(* IEC 61131-3 sources: StandardFunctions/iec61131-st, 18 files *)

(* ---- arithmetic_functions.st ---- *)
(* Definitions of arithmetic functions defined by the IEC61131-3 standard *)

{external}
VAR_GLOBAL
	PI_REAL : REAL;
	PI_LREAL : LREAL;
	FRAC_PI_2_REAL : REAL;
	FRAC_PI_2_LREAL : LREAL;
	FRAC_PI_4_REAL : REAL;
	FRAC_PI_4_LREAL : LREAL;
	E_REAL : REAL;
	E_LREAL : LREAL;
END_VAR

(* Calculates the square root of a given value *)
{external}
FUNCTION SQRT<T : ANY_REAL> : T
VAR_INPUT
	in : T;
END_VAR
END_FUNCTION

(** Logarithmic functions **)

(* Calculates the natural logarithm of the given value *)
{external}
FUNCTION LN<T : ANY_REAL> : T
VAR_INPUT
	in : T;
END_VAR
END_FUNCTION

(* Calculates the base 10 logarithm of the given value *)
{external}
FUNCTION LOG<T : ANY_REAL> : T
VAR_INPUT
	in : T;
END_VAR
END_FUNCTION

(* Calculates the natural exporenent of the given value *)
{external}
FUNCTION EXP<T : ANY_REAL> : T
VAR_INPUT
	in : T;
END_VAR
END_FUNCTION

(** Trigonometric functions **)

(* Calculates the sine of the given value in radiants *)
{external}
FUNCTION SIN<T : ANY_REAL> : T
VAR_INPUT
	rad : T;
END_VAR
END_FUNCTION

(* Calculates the cosine of the given value in radiants *)
{external}
FUNCTION COS<T : ANY_REAL> : T
VAR_INPUT
	rad : T;
END_VAR
END_FUNCTION

(* Calculates the tangent of the given value in radiants *)
{external}
FUNCTION TAN<T : ANY_REAL> : T
VAR_INPUT
	rad : T;
END_VAR
END_FUNCTION

(* Calculates the arc sine of the given value *)
{external}
FUNCTION ASIN<T : ANY_REAL> : T
VAR_INPUT
	in : T;
END_VAR
END_FUNCTION

(* Calculates the arc cosine of the given value *)
{external}
FUNCTION ACOS<T : ANY_REAL> : T
VAR_INPUT
	in : T;
END_VAR
END_FUNCTION

(* Calculates the arc tangent of the given value *)
{external}
FUNCTION ATAN<T : ANY_REAL> : T
VAR_INPUT
	in : T;
END_VAR
END_FUNCTION

(* Calculate the four quadrant arc tangent of the given values *)
{external}
FUNCTION ATAN2<T : ANY_REAL> : T
VAR_INPUT
	y : T;
	x : T;
END_VAR
END_FUNCTION

(* ---- math.st ---- *)
(* Definitions of arithmetic functions defined by the IEC61131-3 standard *)

@EXTERNAL
VAR_GLOBAL
	PI_REAL : REAL;
	PI_LREAL : LREAL;
	FRAC_PI_2_REAL : REAL;
	FRAC_PI_2_LREAL : LREAL;
	FRAC_PI_4_REAL : REAL;
	FRAC_PI_4_LREAL : LREAL;
	E_REAL : REAL;
	E_LREAL : LREAL;
END_VAR

(* Calculates the square root of a given value *)
@EXTERNAL
FUNCTION SQRT<T : ANY_REAL> : T
VAR_INPUT
	in : T;
END_VAR
END_FUNCTION

(** Logarithmic functions **)

(* Calculates the natural logarithm of the given value *)
@EXTERNAL
FUNCTION LN<T : ANY_REAL> : T
VAR_INPUT
	in : T;
END_VAR
END_FUNCTION

(* Calculates the base 10 logarithm of the given value *)
@EXTERNAL
FUNCTION LOG<T : ANY_REAL> : T
VAR_INPUT
	in : T;
END_VAR
END_FUNCTION

(* Calculates the natural exporenent of the given value *)
@EXTERNAL
FUNCTION EXP<T : ANY_REAL> : T
VAR_INPUT
	in : T;
END_VAR
END_FUNCTION

(** Trigonometric functions **)

(* Calculates the sine of the given value in radiants *)
@EXTERNAL
FUNCTION SIN<T : ANY_REAL> : T
VAR_INPUT
	rad : T;
END_VAR
END_FUNCTION

(* Calculates the cosine of the given value in radiants *)
@EXTERNAL
FUNCTION COS<T : ANY_REAL> : T
VAR_INPUT
	rad : T;
END_VAR
END_FUNCTION

(* Calculates the tangent of the given value in radiants *)
@EXTERNAL
FUNCTION TAN<T : ANY_REAL> : T
VAR_INPUT
	rad : T;
END_VAR
END_FUNCTION

(* Calculates the arc sine of the given value *)
@EXTERNAL
FUNCTION ASIN<T : ANY_REAL> : T
VAR_INPUT
	in : T;
END_VAR
END_FUNCTION

(* Calculates the arc cosine of the given value *)
@EXTERNAL
FUNCTION ACOS<T : ANY_REAL> : T
VAR_INPUT
	in : T;
END_VAR
END_FUNCTION

(* Calculates the arc tangent of the given value *)
@EXTERNAL
FUNCTION ATAN<T : ANY_REAL> : T
VAR_INPUT
	in : T;
END_VAR
END_FUNCTION

(* Calculate the four quadrant arc tangent of the given values *)
@EXTERNAL
FUNCTION ATAN2<T : ANY_REAL> : T
VAR_INPUT
	y : T;
	x : T;
END_VAR
END_FUNCTION

(* ---- bit_conversion.st ---- *)
(********************
*
* Converts LWORD to DWORD
*
*********************)
FUNCTION LWORD_TO_DWORD : DWORD
VAR_INPUT
	in : LWORD;
END_VAR
	LWORD_TO_DWORD := in;
END_FUNCTION

(********************
*
* Converts LWORD to WORD
*
*********************)
FUNCTION LWORD_TO_WORD : WORD
VAR_INPUT
	in : LWORD;
END_VAR
	LWORD_TO_WORD := in;
END_FUNCTION

(********************
*
* Converts LWORD to BYTE
*
*********************)
FUNCTION LWORD_TO_BYTE : BYTE
VAR_INPUT
	in : LWORD;
END_VAR
	LWORD_TO_BYTE := in;
END_FUNCTION

(********************
*
* Converts LWORD to BOOL
*
*********************)
FUNCTION LWORD_TO_BOOL : BOOL
VAR_INPUT
	in : LWORD;
END_VAR
	LWORD_TO_BOOL := in;
END_FUNCTION

(********************
*
* Converts DWORD to LWORD
*
*********************)
FUNCTION DWORD_TO_LWORD : LWORD
VAR_INPUT
	in : DWORD;
END_VAR
	DWORD_TO_LWORD := in;
END_FUNCTION

(********************
*
* Converts DWORD to WORD
*
*********************)
FUNCTION DWORD_TO_WORD : WORD
VAR_INPUT
	in : DWORD;
END_VAR
	DWORD_TO_WORD := in;
END_FUNCTION

(********************
*
* Converts DWORD to BYTE
*
*********************)
FUNCTION DWORD_TO_BYTE : BYTE
VAR_INPUT
	in : DWORD;
END_VAR
	DWORD_TO_BYTE := in;
END_FUNCTION

(********************
*
* Converts DWORD to BOOL
*
*********************)
FUNCTION DWORD_TO_BOOL : BOOL
VAR_INPUT
	in : DWORD;
END_VAR
	DWORD_TO_BOOL := in;
END_FUNCTION

(********************
*
* Converts WORD to LWORD
*
*********************)
FUNCTION WORD_TO_LWORD : LWORD
VAR_INPUT
	in : WORD;
END_VAR
	WORD_TO_LWORD := in;
END_FUNCTION

(********************
*
* Converts WORD to DWORD
*
*********************)
FUNCTION WORD_TO_DWORD : DWORD
VAR_INPUT
	in : WORD;
END_VAR
	WORD_TO_DWORD := in;
END_FUNCTION

(********************
*
* Converts WORD to BYTE
*
*********************)
FUNCTION WORD_TO_BYTE : BYTE
VAR_INPUT
	in : WORD;
END_VAR
	WORD_TO_BYTE := in;
END_FUNCTION

(********************
*
* Converts WORD to BOOL
*
*********************)
FUNCTION WORD_TO_BOOL : BOOL
VAR_INPUT
	in : WORD;
END_VAR
	WORD_TO_BOOL := in;
END_FUNCTION

(********************
*
* Converts BYTE to LWORD
*
*********************)
FUNCTION BYTE_TO_LWORD : LWORD
VAR_INPUT
	in : BYTE;
END_VAR
	BYTE_TO_LWORD := in;
END_FUNCTION

(********************
*
* Converts BYTE to DWORD
*
*********************)
FUNCTION BYTE_TO_DWORD : DWORD
VAR_INPUT
	in : BYTE;
END_VAR
	BYTE_TO_DWORD := in;
END_FUNCTION

(********************
*
* Converts BYTE to WORD
*
*********************)
FUNCTION BYTE_TO_WORD : WORD
VAR_INPUT
	in : BYTE;
END_VAR
	BYTE_TO_WORD := in;
END_FUNCTION

(********************
*
* Converts BYTE to BOOL
*
*********************)
FUNCTION BYTE_TO_BOOL : BOOL
VAR_INPUT
	in : BYTE;
END_VAR
	BYTE_TO_BOOL := in;
END_FUNCTION

(********************
*
* Converts BOOL to LWORD
*
*********************)
FUNCTION BOOL_TO_LWORD : LWORD
VAR_INPUT
	in : BOOL;
END_VAR
	BOOL_TO_LWORD := in;
END_FUNCTION

(********************
*
* Converts BOOL to DWORD
*
*********************)
FUNCTION BOOL_TO_DWORD : DWORD
VAR_INPUT
	in : BOOL;
END_VAR
	BOOL_TO_DWORD := in;
END_FUNCTION

(********************
*
* Converts BOOL to WORD
*
*********************)
FUNCTION BOOL_TO_WORD : WORD
VAR_INPUT
	in : BOOL;
END_VAR
	BOOL_TO_WORD := in;
END_FUNCTION

(********************
*
* Converts BOOL to BYTE
*
*********************)
FUNCTION BOOL_TO_BYTE : BYTE
VAR_INPUT
	in : BOOL;
END_VAR
	BOOL_TO_BYTE := in;
END_FUNCTION

(* ---- bit_num_conversion.st ---- *)
(********************
*
* Converts LWORD to LREAL
*
*********************)
FUNCTION LWORD_TO_LREAL : LREAL
VAR_INPUT
	in : LWORD;
END_VAR
	LWORD_TO_LREAL := in;
END_FUNCTION

(********************
*
* Converts LWORD to LINT
*
*********************)
FUNCTION LWORD_TO_LINT : LINT
VAR_INPUT
	in : LWORD;
END_VAR
	LWORD_TO_LINT := in;
END_FUNCTION

(********************
*
* Converts LWORD to DINT
*
*********************)
FUNCTION LWORD_TO_DINT : DINT
VAR_INPUT
	in : LWORD;
END_VAR
	LWORD_TO_DINT := in;
END_FUNCTION

(********************
*
* Converts LWORD to INT
*
*********************)
FUNCTION LWORD_TO_INT : INT
VAR_INPUT
	in : LWORD;
END_VAR
	LWORD_TO_INT := in;
END_FUNCTION

(********************
*
* Converts LWORD to SINT
*
*********************)
FUNCTION LWORD_TO_SINT : SINT
VAR_INPUT
	in : LWORD;
END_VAR
	LWORD_TO_SINT := in;
END_FUNCTION

(********************
*
* Converts LWORD to ULINT
*
*********************)
FUNCTION LWORD_TO_ULINT : ULINT
VAR_INPUT
	in : LWORD;
END_VAR
	LWORD_TO_ULINT := in;
END_FUNCTION

(********************
*
* Converts LWORD to UDINT
*
*********************)
FUNCTION LWORD_TO_UDINT : UDINT
VAR_INPUT
	in : LWORD;
END_VAR
	LWORD_TO_UDINT := in;
END_FUNCTION

(********************
*
* Converts LWORD to UINT
*
*********************)
FUNCTION LWORD_TO_UINT : UINT
VAR_INPUT
	in : LWORD;
END_VAR
	LWORD_TO_UINT := in;
END_FUNCTION

(********************
*
* Converts LWORD to USINT
*
*********************)
FUNCTION LWORD_TO_USINT : USINT
VAR_INPUT
	in : LWORD;
END_VAR
	LWORD_TO_USINT := in;
END_FUNCTION

(********************
*
* Converts DWORD to REAL
*
*********************)
FUNCTION DWORD_TO_REAL : REAL
VAR_INPUT
	in : DWORD;
END_VAR
	DWORD_TO_REAL := in;
END_FUNCTION

(********************
*
* Converts DWORD to LINT
*
*********************)
FUNCTION DWORD_TO_LINT : LINT
VAR_INPUT
	in : DWORD;
END_VAR
	DWORD_TO_LINT := in;
END_FUNCTION

(********************
*
* Converts DWORD to DINT
*
*********************)
FUNCTION DWORD_TO_DINT : DINT
VAR_INPUT
	in : DWORD;
END_VAR
	DWORD_TO_DINT := in;
END_FUNCTION

(********************
*
* Converts DWORD to INT
*
*********************)
FUNCTION DWORD_TO_INT : INT
VAR_INPUT
	in : DWORD;
END_VAR
	DWORD_TO_INT := in;
END_FUNCTION

(********************
*
* Converts DWORD to SINT
*
*********************)
FUNCTION DWORD_TO_SINT : SINT
VAR_INPUT
	in : DWORD;
END_VAR
	DWORD_TO_SINT := in;
END_FUNCTION

(********************
*
* Converts DWORD to ULINT
*
*********************)
FUNCTION DWORD_TO_ULINT : ULINT
VAR_INPUT
	in : DWORD;
END_VAR
	DWORD_TO_ULINT := in;
END_FUNCTION

(********************
*
* Converts DWORD to UDINT
*
*********************)
FUNCTION DWORD_TO_UDINT : UDINT
VAR_INPUT
	in : DWORD;
END_VAR
	DWORD_TO_UDINT := in;
END_FUNCTION

(********************
*
* Converts DWORD to UINT
*
*********************)
FUNCTION DWORD_TO_UINT : UINT
VAR_INPUT
	in : DWORD;
END_VAR
	DWORD_TO_UINT := in;
END_FUNCTION

(********************
*
* Converts DWORD to USINT
*
*********************)
FUNCTION DWORD_TO_USINT : USINT
VAR_INPUT
	in : DWORD;
END_VAR
	DWORD_TO_USINT := in;
END_FUNCTION

(********************
*
* Converts WORD to LINT
*
*********************)
FUNCTION WORD_TO_LINT : LINT
VAR_INPUT
	in : WORD;
END_VAR
	WORD_TO_LINT := in;
END_FUNCTION

(********************
*
* Converts WORD to DINT
*
*********************)
FUNCTION WORD_TO_DINT : DINT
VAR_INPUT
	in : WORD;
END_VAR
	WORD_TO_DINT := in;
END_FUNCTION

(********************
*
* Converts WORD to INT
*
*********************)
FUNCTION WORD_TO_INT : INT
VAR_INPUT
	in : WORD;
END_VAR
	WORD_TO_INT := in;
END_FUNCTION

(********************
*
* Converts WORD to SINT
*
*********************)
FUNCTION WORD_TO_SINT : SINT
VAR_INPUT
	in : WORD;
END_VAR
	WORD_TO_SINT := in;
END_FUNCTION

(********************
*
* Converts WORD to ULINT
*
*********************)
FUNCTION WORD_TO_ULINT : ULINT
VAR_INPUT
	in : WORD;
END_VAR
	WORD_TO_ULINT := in;
END_FUNCTION

(********************
*
* Converts WORD to UDINT
*
*********************)
FUNCTION WORD_TO_UDINT : UDINT
VAR_INPUT
	in : WORD;
END_VAR
	WORD_TO_UDINT := in;
END_FUNCTION

(********************
*
* Converts WORD to UINT
*
*********************)
FUNCTION WORD_TO_UINT : UINT
VAR_INPUT
	in : WORD;
END_VAR
	WORD_TO_UINT := in;
END_FUNCTION

(********************
*
* Converts WORD to USINT
*
*********************)
FUNCTION WORD_TO_USINT : USINT
VAR_INPUT
	in : WORD;
END_VAR
	WORD_TO_USINT := in;
END_FUNCTION

(********************
*
* Converts BYTE to LINT
*
*********************)
FUNCTION BYTE_TO_LINT : LINT
VAR_INPUT
	in : BYTE;
END_VAR
	BYTE_TO_LINT := in;
END_FUNCTION

(********************
*
* Converts BYTE to DINT
*
*********************)
FUNCTION BYTE_TO_DINT : DINT
VAR_INPUT
	in : BYTE;
END_VAR
	BYTE_TO_DINT := in;
END_FUNCTION

(********************
*
* Converts BYTE to INT
*
*********************)
FUNCTION BYTE_TO_INT : INT
VAR_INPUT
	in : BYTE;
END_VAR
	BYTE_TO_INT := in;
END_FUNCTION

(********************
*
* Converts BYTE to SINT
*
*********************)
FUNCTION BYTE_TO_SINT : SINT
VAR_INPUT
	in : BYTE;
END_VAR
	BYTE_TO_SINT := in;
END_FUNCTION

(********************
*
* Converts BYTE to ULINT
*
*********************)
FUNCTION BYTE_TO_ULINT : ULINT
VAR_INPUT
	in : BYTE;
END_VAR
	BYTE_TO_ULINT := in;
END_FUNCTION

(********************
*
* Converts BYTE to UDINT
*
*********************)
FUNCTION BYTE_TO_UDINT : UDINT
VAR_INPUT
	in : BYTE;
END_VAR
	BYTE_TO_UDINT := in;
END_FUNCTION

(********************
*
* Converts BYTE to UINT
*
*********************)
FUNCTION BYTE_TO_UINT : UINT
VAR_INPUT
	in : BYTE;
END_VAR
	BYTE_TO_UINT := in;
END_FUNCTION

(********************
*
* Converts BYTE to USINT
*
*********************)
FUNCTION BYTE_TO_USINT : USINT
VAR_INPUT
	in : BYTE;
END_VAR
	BYTE_TO_USINT := in;
END_FUNCTION

(********************
*
* Converts BOOL to LINT
*
*********************)
FUNCTION BOOL_TO_LINT : LINT
VAR_INPUT
	in : BOOL;
END_VAR
	BOOL_TO_LINT := in;
END_FUNCTION

(********************
*
* Converts BOOL to DINT
*
*********************)
FUNCTION BOOL_TO_DINT : DINT
VAR_INPUT
	in : BOOL;
END_VAR
	BOOL_TO_DINT := in;
END_FUNCTION

(********************
*
* Converts BOOL to INT
*
*********************)
FUNCTION BOOL_TO_INT : INT
VAR_INPUT
	in : BOOL;
END_VAR
	BOOL_TO_INT := in;
END_FUNCTION

(********************
*
* Converts BOOL to SINT
*
*********************)
FUNCTION BOOL_TO_SINT : SINT
VAR_INPUT
	in : BOOL;
END_VAR
	BOOL_TO_SINT := in;
END_FUNCTION

(********************
*
* Converts BOOL to ULINT
*
*********************)
FUNCTION BOOL_TO_ULINT : ULINT
VAR_INPUT
	in : BOOL;
END_VAR
	BOOL_TO_ULINT := in;
END_FUNCTION

(********************
*
* Converts BOOL to UDINT
*
*********************)
FUNCTION BOOL_TO_UDINT : UDINT
VAR_INPUT
	in : BOOL;
END_VAR
	BOOL_TO_UDINT := in;
END_FUNCTION

(********************
*
* Converts BOOL to UINT
*
*********************)
FUNCTION BOOL_TO_UINT : UINT
VAR_INPUT
	in : BOOL;
END_VAR
	BOOL_TO_UINT := in;
END_FUNCTION

(********************
*
* Converts BOOL to USINT
*
*********************)
FUNCTION BOOL_TO_USINT : USINT
VAR_INPUT
	in : BOOL;
END_VAR
	BOOL_TO_USINT := in;
END_FUNCTION

(********************
*
* Converts LREAL to LWORD
*
*********************)
FUNCTION LREAL_TO_LWORD : LWORD
VAR_INPUT
	in : LREAL;
END_VAR
	LREAL_TO_LWORD := in;
END_FUNCTION

(********************
*
* Converts REAL to DWORD
*
*********************)
FUNCTION REAL_TO_DWORD : DWORD
VAR_INPUT
	in : REAL;
END_VAR
	REAL_TO_DWORD := in;
END_FUNCTION

(********************
*
* Converts LINT to LWORD
*
*********************)
FUNCTION LINT_TO_LWORD : LWORD
VAR_INPUT
	in : LINT;
END_VAR
	LINT_TO_LWORD := in;
END_FUNCTION

(********************
*
* Converts LINT to DWORD
*
*********************)
FUNCTION LINT_TO_DWORD : DWORD
VAR_INPUT
	in : LINT;
END_VAR
	LINT_TO_DWORD := in;
END_FUNCTION

(********************
*
* Converts LINT to WORD
*
*********************)
FUNCTION LINT_TO_WORD : WORD
VAR_INPUT
	in : LINT;
END_VAR
	LINT_TO_WORD := in;
END_FUNCTION

(********************
*
* Converts LINT to BYTE
*
*********************)
FUNCTION LINT_TO_BYTE : BYTE
VAR_INPUT
	in : LINT;
END_VAR
	LINT_TO_BYTE := in;
END_FUNCTION

(********************
*
* Converts DINT to LWORD
*
*********************)
FUNCTION DINT_TO_LWORD : LWORD
VAR_INPUT
	in : DINT;
END_VAR
	DINT_TO_LWORD := in;
END_FUNCTION

(********************
*
* Converts DINT to DWORD
*
*********************)
FUNCTION DINT_TO_DWORD : DWORD
VAR_INPUT
	in : DINT;
END_VAR
	DINT_TO_DWORD := in;
END_FUNCTION

(********************
*
* Converts DINT to WORD
*
*********************)
FUNCTION DINT_TO_WORD : WORD
VAR_INPUT
	in : DINT;
END_VAR
	DINT_TO_WORD := in;
END_FUNCTION

(********************
*
* Converts DINT to BYTE
*
*********************)
FUNCTION DINT_TO_BYTE : BYTE
VAR_INPUT
	in : DINT;
END_VAR
	DINT_TO_BYTE := in;
END_FUNCTION

(********************
*
* Converts INT to LWORD
*
*********************)
FUNCTION INT_TO_LWORD : LWORD
VAR_INPUT
	in : INT;
END_VAR
	INT_TO_LWORD := in;
END_FUNCTION

(********************
*
* Converts INT to DWORD
*
*********************)
FUNCTION INT_TO_DWORD : DWORD
VAR_INPUT
	in : INT;
END_VAR
	INT_TO_DWORD := in;
END_FUNCTION

(********************
*
* Converts INT to WORD
*
*********************)
FUNCTION INT_TO_WORD : WORD
VAR_INPUT
	in : INT;
END_VAR
	INT_TO_WORD := in;
END_FUNCTION

(********************
*
* Converts INT to BYTE
*
*********************)
FUNCTION INT_TO_BYTE : BYTE
VAR_INPUT
	in : INT;
END_VAR
	INT_TO_BYTE := in;
END_FUNCTION

(********************
*
* Converts SINT to LWORD
*
*********************)
FUNCTION SINT_TO_LWORD : LWORD
VAR_INPUT
	in : SINT;
END_VAR
	SINT_TO_LWORD := in;
END_FUNCTION

(********************
*
* Converts SINT to DWORD
*
*********************)
FUNCTION SINT_TO_DWORD : DWORD
VAR_INPUT
	in : SINT;
END_VAR
	SINT_TO_DWORD := in;
END_FUNCTION

(********************
*
* Converts SINT to WORD
*
*********************)
FUNCTION SINT_TO_WORD : WORD
VAR_INPUT
	in : SINT;
END_VAR
	SINT_TO_WORD := in;
END_FUNCTION

(********************
*
* Converts SINT to BYTE
*
*********************)
FUNCTION SINT_TO_BYTE : BYTE
VAR_INPUT
	in : SINT;
END_VAR
	SINT_TO_BYTE := in;
END_FUNCTION

(********************
*
* Converts ULINT to LWORD
*
*********************)
FUNCTION ULINT_TO_LWORD : LWORD
VAR_INPUT
	in : ULINT;
END_VAR
	ULINT_TO_LWORD := in;
END_FUNCTION

(********************
*
* Converts ULINT to DWORD
*
*********************)
FUNCTION ULINT_TO_DWORD : DWORD
VAR_INPUT
	in : ULINT;
END_VAR
	ULINT_TO_DWORD := in;
END_FUNCTION

(********************
*
* Converts ULINT to WORD
*
*********************)
FUNCTION ULINT_TO_WORD : WORD
VAR_INPUT
	in : ULINT;
END_VAR
	ULINT_TO_WORD := in;
END_FUNCTION

(********************
*
* Converts ULINT to BYTE
*
*********************)
FUNCTION ULINT_TO_BYTE : BYTE
VAR_INPUT
	in : ULINT;
END_VAR
	ULINT_TO_BYTE := in;
END_FUNCTION

(********************
*
* Converts UDINT to LWORD
*
*********************)
FUNCTION UDINT_TO_LWORD : LWORD
VAR_INPUT
	in : UDINT;
END_VAR
	UDINT_TO_LWORD := in;
END_FUNCTION

(********************
*
* Converts UDINT to DWORD
*
*********************)
FUNCTION UDINT_TO_DWORD : DWORD
VAR_INPUT
	in : UDINT;
END_VAR
	UDINT_TO_DWORD := in;
END_FUNCTION

(********************
*
* Converts UDINT to WORD
*
*********************)
FUNCTION UDINT_TO_WORD : WORD
VAR_INPUT
	in : UDINT;
END_VAR
	UDINT_TO_WORD := in;
END_FUNCTION

(********************
*
* Converts UDINT to BYTE
*
*********************)
FUNCTION UDINT_TO_BYTE : BYTE
VAR_INPUT
	in : UDINT;
END_VAR
	UDINT_TO_BYTE := in;
END_FUNCTION

(********************
*
* Converts UINT to LWORD
*
*********************)
FUNCTION UINT_TO_LWORD : LWORD
VAR_INPUT
	in : UINT;
END_VAR
	UINT_TO_LWORD := in;
END_FUNCTION

(********************
*
* Converts UINT to DWORD
*
*********************)
FUNCTION UINT_TO_DWORD : DWORD
VAR_INPUT
	in : UINT;
END_VAR
	UINT_TO_DWORD := in;
END_FUNCTION

(********************
*
* Converts UINT to WORD
*
*********************)
FUNCTION UINT_TO_WORD : WORD
VAR_INPUT
	in : UINT;
END_VAR
	UINT_TO_WORD := in;
END_FUNCTION

(********************
*
* Converts UINT to BYTE
*
*********************)
FUNCTION UINT_TO_BYTE : BYTE
VAR_INPUT
	in : UINT;
END_VAR
	UINT_TO_BYTE := in;
END_FUNCTION

(********************
*
* Converts USINT to LWORD
*
*********************)
FUNCTION USINT_TO_LWORD : LWORD
VAR_INPUT
	in : USINT;
END_VAR
	USINT_TO_LWORD := in;
END_FUNCTION

(********************
*
* Converts USINT to DWORD
*
*********************)
FUNCTION USINT_TO_DWORD : DWORD
VAR_INPUT
	in : USINT;
END_VAR
	USINT_TO_DWORD := in;
END_FUNCTION

(********************
*
* Converts USINT to WORD
*
*********************)
FUNCTION USINT_TO_WORD : WORD
VAR_INPUT
	in : USINT;
END_VAR
	USINT_TO_WORD := in;
END_FUNCTION

(********************
*
* Converts USINT to BYTE
*
*********************)
FUNCTION USINT_TO_BYTE : BYTE
VAR_INPUT
	in : USINT;
END_VAR
	USINT_TO_BYTE := in;
END_FUNCTION

(* ---- date_time_conversion.st ---- *)
(********************
*
* Converts DT/LDT to DATE
*
*********************)
@EXTERNAL
FUNCTION DATE_AND_TIME_TO_DATE : DATE
VAR_INPUT
	in : DT;
END_VAR
END_FUNCTION

(********************
*
* Converts DT/LDT to TOD/LTOD
*
*********************)
@EXTERNAL
FUNCTION DATE_AND_TIME_TO_TIME_OF_DAY : TOD
VAR_INPUT
	in : DT;
END_VAR
END_FUNCTION

(********************
*
* Converts LTIME to TIME
*
*********************)
FUNCTION LTIME_TO_TIME : TIME
VAR_INPUT
	in : LTIME;
END_VAR
	LTIME_TO_TIME := in;
END_FUNCTION

(********************
*
* Converts TIME to LTIME
*
*********************)
FUNCTION TIME_TO_LTIME : LTIME
VAR_INPUT
	in : TIME;
END_VAR
	TIME_TO_LTIME := in;
END_FUNCTION

(********************
*
* Converts LDT to DT
*
*********************)
FUNCTION LDT_TO_DT : DT
VAR_INPUT
	in : LDT;
END_VAR
	LDT_TO_DT := in;
END_FUNCTION

(********************
*
* Converts LDT to DATE
*
*********************)
FUNCTION LDT_TO_DATE : DATE
VAR_INPUT
	in : LDT;
END_VAR
	LDT_TO_DATE := DATE_AND_TIME_TO_DATE(in);
END_FUNCTION

(********************
*
* Converts LDT to LTOD
*
*********************)
FUNCTION LDT_TO_LTOD : LTOD
VAR_INPUT
	in : LDT;
END_VAR
	LDT_TO_LTOD := DATE_AND_TIME_TO_TIME_OF_DAY(in);
END_FUNCTION

(********************
*
* Converts LDT to TOD
*
*********************)
FUNCTION LDT_TO_TOD : TOD
VAR_INPUT
	in : LDT;
END_VAR
	LDT_TO_TOD := DATE_AND_TIME_TO_TIME_OF_DAY(in);
END_FUNCTION

(********************
*
* Converts DT to LDT
*
*********************)
FUNCTION DT_TO_LDT : LDT
VAR_INPUT
	in : DT;
END_VAR
	DT_TO_LDT := in;
END_FUNCTION

(********************
*
* Converts DT to DATE
*
*********************)
FUNCTION DT_TO_DATE : DATE
VAR_INPUT
	in : DT;
END_VAR
	DT_TO_DATE := DATE_AND_TIME_TO_DATE(in);
END_FUNCTION

(********************
*
* Converts DT to LTOD
*
*********************)
FUNCTION DT_TO_LTOD : LTOD
VAR_INPUT
	in : DT;
END_VAR
	DT_TO_LTOD := DATE_AND_TIME_TO_TIME_OF_DAY(in);
END_FUNCTION

(********************
*
* Converts DT to TOD
*
*********************)
FUNCTION DT_TO_TOD : TOD
VAR_INPUT
	in : DT;
END_VAR
	DT_TO_TOD := DATE_AND_TIME_TO_TIME_OF_DAY(in);
END_FUNCTION

(********************
*
* Converts LTOD to TOD
*
*********************)
FUNCTION LTOD_TO_TOD : TOD
VAR_INPUT
	in : LTOD;
END_VAR
	LTOD_TO_TOD := in;
END_FUNCTION

(********************
*
* Converts TOD to LTOD
*
*********************)
FUNCTION TOD_TO_LTOD : LTOD
VAR_INPUT
	in : TOD;
END_VAR
	TOD_TO_LTOD := in;
END_FUNCTION

(* ---- date_time_numeric_functions.st ---- *)
(********************
*
* This operator returns the value of adding up the operands.
*
*********************)
FUNCTION ADD <T1: ANY, T2: ANY> : T1
VAR_INPUT
	IN1 : T1;
	IN2 : T2;
END_VAR
END_FUNCTION

(* Specialized implementation of ADD for TIME *)
FUNCTION ADD__TIME__TIME : TIME
VAR_INPUT
	IN1 : TIME;
	IN2 : TIME;
END_VAR
	ADD__TIME__TIME := ADD_TIME(IN1, IN2);
END_FUNCTION

(********************
*
* This operator returns the value of adding up two TIME operands.
*
*********************)
@EXTERNAL
FUNCTION ADD_TIME : TIME
VAR_INPUT
	IN1 : TIME;
	IN2 : TIME;
END_VAR
END_FUNCTION

(********************
*
* This operator returns the value of adding up two LTIME operands.
*
*********************)
FUNCTION ADD_LTIME : LTIME
VAR_INPUT
	IN1 : LTIME;
	IN2 : LTIME;
END_VAR
	ADD_LTIME := ADD_TIME(IN1, IN2);
END_FUNCTION

(* Specialized implementation of ADD for TOD *)
FUNCTION ADD__TIME_OF_DAY__TIME : TOD
VAR_INPUT
	IN1 : TOD;
	IN2 : TIME;
END_VAR
	ADD__TIME_OF_DAY__TIME := ADD_TOD_TIME(IN1, IN2);
END_FUNCTION

(********************
*
* This operator returns the value of adding up TOD and TIME.
* If the result overflows 0 will be returned
*
*********************)
@EXTERNAL
FUNCTION ADD_TOD_TIME : TOD
VAR_INPUT
	IN1 : TOD;
	IN2 : TIME;
END_VAR
END_FUNCTION

(********************
*
* This operator returns the value of adding up LTOD and LTIME.
* If the result overflows 0 will be returned
*
*********************)
FUNCTION ADD_LTOD_LTIME : LTOD
VAR_INPUT
	IN1 : LTOD;
	IN2 : LTIME;
END_VAR
	ADD_LTOD_LTIME := ADD_TOD_TIME(IN1, IN2);
END_FUNCTION

(* Specialized implementation of ADD for DT *)
FUNCTION ADD__DATE_AND_TIME__TIME : DT
VAR_INPUT
	IN1 : DT;
	IN2 : TIME;
END_VAR
	ADD__DATE_AND_TIME__TIME := ADD_DT_TIME(IN1, IN2);
END_FUNCTION

(********************
*
* This operator returns the value of adding up DT and TIME.
* If the result overflows 0 will be returned
*
*********************)
@EXTERNAL
FUNCTION ADD_DT_TIME : DT
VAR_INPUT
	IN1 : DT;
	IN2 : TIME;
END_VAR
END_FUNCTION

(********************
*
* This operator returns the value of adding up LDT and LTIME.
* If the result overflows 0 will be returned
*
*********************)
FUNCTION ADD_LDT_LTIME : LDT
VAR_INPUT
	IN1 : LDT;
	IN2 : LTIME;
END_VAR
	ADD_LDT_LTIME := ADD_DT_TIME(IN1, IN2);
END_FUNCTION

(********************
*
* This operator produces the subtraction of the operands.
*
*********************)
FUNCTION SUB <T1: ANY, T2: ANY> : T1
VAR_INPUT
	IN1 : T1;
	IN2 : T2;
END_VAR
END_FUNCTION

(* Specialized implementation of SUB for TIME *)
FUNCTION SUB__TIME__TIME : TIME
VAR_INPUT
	IN1 : TIME;
	IN2 : TIME;
END_VAR
	SUB__TIME__TIME := SUB_TIME(IN1, IN2);
END_FUNCTION

(********************
*
* This operator produces the subtraction of two TIME operands
*
*********************)
@EXTERNAL
FUNCTION SUB_TIME : TIME
VAR_INPUT
	IN1 : TIME;
	IN2 : TIME;
END_VAR
END_FUNCTION

(********************
*
* This operator produces the subtraction of two LTIME operands
*
*********************)
FUNCTION SUB_LTIME : LTIME
VAR_INPUT
	IN1 : LTIME;
	IN2 : LTIME;
END_VAR
	SUB_LTIME := SUB_TIME(IN1, IN2);
END_FUNCTION

(* Specialized implementation of SUB for DATE *)
FUNCTION SUB__DATE__DATE : TIME
VAR_INPUT
	IN1 : DATE;
	IN2 : DATE;
END_VAR
	SUB__DATE__DATE := SUB_DATE_DATE(IN1, IN2);
END_FUNCTION

(********************
*
* This operator produces the subtraction of two DATE operands returning TIME
* If the result overflows 0 will be returned
*
*********************)
@EXTERNAL
FUNCTION SUB_DATE_DATE : TIME
VAR_INPUT
	IN1 : DATE;
	IN2 : DATE;
END_VAR
END_FUNCTION

(********************
*
* This operator produces the subtraction of two LDATE operands returning LTIME
* If the result overflows 0 will be returned
*
*********************)
FUNCTION SUB_LDATE_LDATE : LTIME
VAR_INPUT
	IN1 : LDATE;
	IN2 : LDATE;
END_VAR
	SUB_LDATE_LDATE := SUB_DATE_DATE(IN1, IN2);
END_FUNCTION

(* Specialized implementation of SUB for TOD and TIME *)
FUNCTION SUB__TIME_OF_DAY__TIME : TOD
VAR_INPUT
	IN1 : TOD;
	IN2 : TIME;
END_VAR
	SUB__TIME_OF_DAY__TIME := SUB_TOD_TIME(IN1, IN2);
END_FUNCTION

(********************
*
* This operator produces the subtraction of TOD and TIME returning TOD
* If the result overflows 0 will be returned
*
*********************)
@EXTERNAL
FUNCTION SUB_TOD_TIME : TOD
VAR_INPUT
	IN1 : TOD;
	IN2 : TIME;
END_VAR
END_FUNCTION

(********************
*
* This operator produces the subtraction of LTOD and LTIME returning LTOD
* If the result overflows 0 will be returned
*
*********************)
FUNCTION SUB_LTOD_LTIME : LTOD
VAR_INPUT
	IN1 : LTOD;
	IN2 : LTIME;
END_VAR
	SUB_LTOD_LTIME := SUB_TOD_TIME(IN1, IN2);
END_FUNCTION

(* Specialized implementation of SUB for TOD *)
FUNCTION SUB__TIME_OF_DAY__TIME_OF_DAY : TIME
VAR_INPUT
	IN1 : TOD;
	IN2 : TOD;
END_VAR
	SUB__TIME_OF_DAY__TIME_OF_DAY := SUB_TOD_TOD(IN1, IN2);
END_FUNCTION

(********************
*
* This operator produces the subtraction of two TOD operands returning TIME
* If the result overflows 0 will be returned
*
*********************)
@EXTERNAL
FUNCTION SUB_TOD_TOD : TIME
VAR_INPUT
	IN1 : TOD;
	IN2 : TOD;
END_VAR
END_FUNCTION

(********************
*
* This operator produces the subtraction of two LTOD operands returning LTIME
* If the result overflows 0 will be returned
*
*********************)
FUNCTION SUB_LTOD_LTOD : LTIME
VAR_INPUT
	IN1 : LTOD;
	IN2 : LTOD;
END_VAR
	SUB_LTOD_LTOD := SUB_TOD_TOD(IN1, IN2);
END_FUNCTION

(* Specialized implementation of SUB for DT and TIME *)
FUNCTION SUB__DATE_AND_TIME__TIME : DT
VAR_INPUT
	IN1 : DT;
	IN2 : TIME;
END_VAR
	SUB__DATE_AND_TIME__TIME := SUB_DT_TIME(IN1, IN2);
END_FUNCTION

(********************
*
* This operator produces the subtraction of DT and TIME returning DT
* If the result overflows 0 will be returned
*
*********************)
@EXTERNAL
FUNCTION SUB_DT_TIME : DT
VAR_INPUT
	IN1 : DT;
	IN2 : TIME;
END_VAR
END_FUNCTION

(********************
*
* This operator produces the subtraction of LDT and LTIME returning LDT
* If the result overflows 0 will be returned
*
*********************)
FUNCTION SUB_LDT_LTIME : LDT
VAR_INPUT
	IN1 : LDT;
	IN2 : LTIME;
END_VAR
	SUB_LDT_LTIME := SUB_DT_TIME(IN1, IN2);
END_FUNCTION

(* Specialized implementation of SUB for DT *)
FUNCTION SUB__DATE_AND_TIME__DATE_AND_TIME : TIME
VAR_INPUT
	IN1 : DT;
	IN2 : DT;
END_VAR
	SUB__DATE_AND_TIME__DATE_AND_TIME := SUB_DT_DT(IN1, IN2);
END_FUNCTION

(********************
*
* This operator produces the subtraction of two DT operands returning TIME
* If the result overflows 0 will be returned
*
*********************)
@EXTERNAL
FUNCTION SUB_DT_DT : TIME
VAR_INPUT
	IN1 : DT;
	IN2 : DT;
END_VAR
END_FUNCTION

(********************
*
* This operator produces the subtraction of two LDT operands returning LTIME
* If the result overflows 0 will be returned
*
*********************)
FUNCTION SUB_LDT_LDT : LTIME
VAR_INPUT
	IN1 : LDT;
	IN2 : LDT;
END_VAR
	SUB_LDT_LDT := SUB_DT_DT(IN1, IN2);
END_FUNCTION

(********************
*
* This operator produces the multiplication of the operands.
*
*********************)
FUNCTION MUL <T1: ANY, T2: ANY> : T1
VAR_INPUT
	IN1 : T1;
	IN2 : T2;
END_VAR
END_FUNCTION

(* Specialized implementation of MUL for TIME and SINT *)
FUNCTION MUL__TIME__SINT : TIME
VAR_INPUT
	IN1 : TIME;
	IN2 : SINT;
END_VAR
	MUL__TIME__SINT := CHECKED_MUL_SIGNED(IN1, IN2);
END_FUNCTION

(* Specialized implementation of MUL for TIME and INT *)
FUNCTION MUL__TIME__INT : TIME
VAR_INPUT
	IN1 : TIME;
	IN2 : INT;
END_VAR
	MUL__TIME__INT := CHECKED_MUL_SIGNED(IN1, IN2);
END_FUNCTION

(* Specialized implementation of MUL for TIME and DINT *)
FUNCTION MUL__TIME__DINT : TIME
VAR_INPUT
	IN1 : TIME;
	IN2 : DINT;
END_VAR
	MUL__TIME__DINT := CHECKED_MUL_SIGNED(IN1, IN2);
END_FUNCTION

(* Specialized implementation of MUL for TIME and LINT *)
FUNCTION MUL__TIME__LINT : TIME
VAR_INPUT
	IN1 : TIME;
	IN2 : LINT;
END_VAR
	MUL__TIME__LINT := CHECKED_MUL_SIGNED(IN1, IN2);
END_FUNCTION

(********************
*
* This operator produces the multiplication of TIME with ANY_SIGNED integer
* If the result overflows 0 will be returned
*
*********************)
@EXTERNAL
FUNCTION CHECKED_MUL_SIGNED : TIME
VAR_INPUT
	IN1 : TIME;
	IN2 : LINT;
END_VAR
END_FUNCTION

(* Specialized implementation of MUL for TIME and USINT *)
FUNCTION MUL__TIME__USINT : TIME
VAR_INPUT
	IN1 : TIME;
	IN2 : USINT;
END_VAR
	MUL__TIME__USINT := CHECKED_MUL_UNSIGNED(IN1, IN2);
END_FUNCTION

(* Specialized implementation of MUL for TIME and UINT *)
FUNCTION MUL__TIME__UINT : TIME
VAR_INPUT
	IN1 : TIME;
	IN2 : UINT;
END_VAR
	MUL__TIME__UINT := CHECKED_MUL_UNSIGNED(IN1, IN2);
END_FUNCTION

(* Specialized implementation of MUL for TIME and UDINT *)
FUNCTION MUL__TIME__UDINT : TIME
VAR_INPUT
	IN1 : TIME;
	IN2 : UDINT;
END_VAR
	MUL__TIME__UDINT := CHECKED_MUL_UNSIGNED(IN1, IN2);
END_FUNCTION

(* Specialized implementation of MUL for TIME and ULINT *)
FUNCTION MUL__TIME__ULINT : TIME
VAR_INPUT
	IN1 : TIME;
	IN2 : ULINT;
END_VAR
	MUL__TIME__ULINT := CHECKED_MUL_UNSIGNED(IN1, IN2);
END_FUNCTION

(********************
*
* This operator produces the multiplication of TIME with ANY_UNSIGNED integer
* If the result overflows 0 will be returned
*
*********************)
@EXTERNAL
FUNCTION CHECKED_MUL_UNSIGNED : TIME
VAR_INPUT
	IN1 : TIME;
	IN2 : ULINT;
END_VAR
END_FUNCTION

(********************
*
* This operator produces the multiplication of TIME and ANY_NUM.
*
*********************)
FUNCTION MUL_TIME <T: ANY_NUM> : TIME
VAR_INPUT
	IN1 : TIME;
	IN2 : T;
END_VAR
END_FUNCTION

(* Specialized implementation of MUL_TIME for SINT *)
FUNCTION MUL_TIME__SINT : TIME
VAR_INPUT
	IN1 : TIME;
	IN2 : SINT;
END_VAR
	MUL_TIME__SINT := CHECKED_MUL_SIGNED(IN1, IN2);
END_FUNCTION

(* Specialized implementation of MUL_TIME for INT *)
FUNCTION MUL_TIME__INT : TIME
VAR_INPUT
	IN1 : TIME;
	IN2 : INT;
END_VAR
	MUL_TIME__INT := CHECKED_MUL_SIGNED(IN1, IN2);
END_FUNCTION

(* Specialized implementation of MUL_TIME for DINT *)
FUNCTION MUL_TIME__DINT : TIME
VAR_INPUT
	IN1 : TIME;
	IN2 : DINT;
END_VAR
	MUL_TIME__DINT := CHECKED_MUL_SIGNED(IN1, IN2);
END_FUNCTION

(* Specialized implementation of MUL_TIME for LINT *)
FUNCTION MUL_TIME__LINT : TIME
VAR_INPUT
	IN1 : TIME;
	IN2 : LINT;
END_VAR
	MUL_TIME__LINT := CHECKED_MUL_SIGNED(IN1, IN2);
END_FUNCTION

(* Specialized implementation of MUL_TIME for USINT *)
FUNCTION MUL_TIME__USINT : TIME
VAR_INPUT
	IN1 : TIME;
	IN2 : USINT;
END_VAR
	MUL_TIME__USINT := CHECKED_MUL_UNSIGNED(IN1, IN2);
END_FUNCTION

(* Specialized implementation of MUL_TIME for UINT *)
FUNCTION MUL_TIME__UINT : TIME
VAR_INPUT
	IN1 : TIME;
	IN2 : UINT;
END_VAR
	MUL_TIME__UINT := CHECKED_MUL_UNSIGNED(IN1, IN2);
END_FUNCTION

(* Specialized implementation of MUL_TIME for UDINT *)
FUNCTION MUL_TIME__UDINT : TIME
VAR_INPUT
	IN1 : TIME;
	IN2 : UDINT;
END_VAR
	MUL_TIME__UDINT := CHECKED_MUL_UNSIGNED(IN1, IN2);
END_FUNCTION

(* Specialized implementation of MUL_TIME for ULINT *)
FUNCTION MUL_TIME__ULINT : TIME
VAR_INPUT
	IN1 : TIME;
	IN2 : ULINT;
END_VAR
	MUL_TIME__ULINT := CHECKED_MUL_UNSIGNED(IN1, IN2);
END_FUNCTION

(********************
*
* This operator produces the multiplication of LTIME and ANY_NUM.
*
*********************)
FUNCTION MUL_LTIME <T: ANY_NUM> : LTIME
VAR_INPUT
	IN1 : LTIME;
	IN2 : T;
END_VAR
END_FUNCTION

(* Specialized implementation of MUL_LTIME for SINT *)
FUNCTION MUL_LTIME__SINT : LTIME
VAR_INPUT
	IN1 : LTIME;
	IN2 : SINT;
END_VAR
	MUL_LTIME__SINT := CHECKED_MUL_SIGNED(IN1, IN2);
END_FUNCTION

(* Specialized implementation of MUL_LTIME for INT *)
FUNCTION MUL_LTIME__INT : LTIME
VAR_INPUT
	IN1 : LTIME;
	IN2 : INT;
END_VAR
	MUL_LTIME__INT := CHECKED_MUL_SIGNED(IN1, IN2);
END_FUNCTION

(* Specialized implementation of MUL_LTIME for DINT *)
FUNCTION MUL_LTIME__DINT : LTIME
VAR_INPUT
	IN1 : LTIME;
	IN2 : DINT;
END_VAR
	MUL_LTIME__DINT := CHECKED_MUL_SIGNED(IN1, IN2);
END_FUNCTION

(* Specialized implementation of MUL_LTIME for LINT *)
FUNCTION MUL_LTIME__LINT : LTIME
VAR_INPUT
	IN1 : LTIME;
	IN2 : LINT;
END_VAR
	MUL_LTIME__LINT := CHECKED_MUL_SIGNED(IN1, IN2);
END_FUNCTION

(* Specialized implementation of MUL_LTIME for USINT *)
FUNCTION MUL_LTIME__USINT : LTIME
VAR_INPUT
	IN1 : LTIME;
	IN2 : USINT;
END_VAR
	MUL_LTIME__USINT := CHECKED_MUL_UNSIGNED(IN1, IN2);
END_FUNCTION

(* Specialized implementation of MUL_LTIME for UINT *)
FUNCTION MUL_LTIME__UINT : LTIME
VAR_INPUT
	IN1 : LTIME;
	IN2 : UINT;
END_VAR
	MUL_LTIME__UINT := CHECKED_MUL_UNSIGNED(IN1, IN2);
END_FUNCTION

(* Specialized implementation of MUL_LTIME for UDINT *)
FUNCTION MUL_LTIME__UDINT : LTIME
VAR_INPUT
	IN1 : LTIME;
	IN2 : UDINT;
END_VAR
	MUL_LTIME__UDINT := CHECKED_MUL_UNSIGNED(IN1, IN2);
END_FUNCTION

(* Specialized implementation of MUL_LTIME for ULINT *)
FUNCTION MUL_LTIME__ULINT : LTIME
VAR_INPUT
	IN1 : LTIME;
	IN2 : ULINT;
END_VAR
	MUL_LTIME__ULINT := CHECKED_MUL_UNSIGNED(IN1, IN2);
END_FUNCTION

(********************
*
* This operator produces the division of the operands.
*
*********************)
FUNCTION DIV <T1: ANY, T2: ANY> : T1
VAR_INPUT
	IN1 : T1;
	IN2 : T2;
END_VAR
END_FUNCTION

(* Specialized implementation of DIV for TIME and SINT *)
FUNCTION DIV__TIME__SINT : TIME
VAR_INPUT
	IN1 : TIME;
	IN2 : SINT;
END_VAR
	DIV__TIME__SINT := CHECKED_DIV_SIGNED(IN1, IN2);
END_FUNCTION

(* Specialized implementation of DIV for TIME and INT *)
FUNCTION DIV__TIME__INT : TIME
VAR_INPUT
	IN1 : TIME;
	IN2 : INT;
END_VAR
	DIV__TIME__INT := CHECKED_DIV_SIGNED(IN1, IN2);
END_FUNCTION

(* Specialized implementation of DIV for TIME and DINT *)
FUNCTION DIV__TIME__DINT : TIME
VAR_INPUT
	IN1 : TIME;
	IN2 : DINT;
END_VAR
	DIV__TIME__DINT := CHECKED_DIV_SIGNED(IN1, IN2);
END_FUNCTION

(* Specialized implementation of DIV for TIME and LINT *)
FUNCTION DIV__TIME__LINT : TIME
VAR_INPUT
	IN1 : TIME;
	IN2 : LINT;
END_VAR
	DIV__TIME__LINT := CHECKED_DIV_SIGNED(IN1, IN2);
END_FUNCTION

(********************
*
* This operator produces the division of TIME with ANY_SIGNED integer
* If the result overflows 0 will be returned
* Division by 0 will also return 0
*
*********************)
@EXTERNAL
FUNCTION CHECKED_DIV_SIGNED : TIME
VAR_INPUT
	IN1 : TIME;
	IN2 : LINT;
END_VAR
END_FUNCTION

(* Specialized implementation of DIV for TIME and USINT *)
FUNCTION DIV__TIME__USINT : TIME
VAR_INPUT
	IN1 : TIME;
	IN2 : USINT;
END_VAR
	DIV__TIME__USINT := CHECKED_DIV_UNSIGNED(IN1, IN2);
END_FUNCTION

(* Specialized implementation of DIV for TIME and UINT *)
FUNCTION DIV__TIME__UINT : TIME
VAR_INPUT
	IN1 : TIME;
	IN2 : UINT;
END_VAR
	DIV__TIME__UINT := CHECKED_DIV_UNSIGNED(IN1, IN2);
END_FUNCTION

(* Specialized implementation of DIV for TIME and UDINT *)
FUNCTION DIV__TIME__UDINT : TIME
VAR_INPUT
	IN1 : TIME;
	IN2 : UDINT;
END_VAR
	DIV__TIME__UDINT := CHECKED_DIV_UNSIGNED(IN1, IN2);
END_FUNCTION

(* Specialized implementation of DIV for TIME and ULINT *)
FUNCTION DIV__TIME__ULINT : TIME
VAR_INPUT
	IN1 : TIME;
	IN2 : ULINT;
END_VAR
	DIV__TIME__ULINT := CHECKED_DIV_UNSIGNED(IN1, IN2);
END_FUNCTION

(********************
*
* This operator produces the division of TIME with ANY_UNSIGNED integer
* If the result overflows 0 will be returned
* Division by 0 will also return 0
*
*********************)
@EXTERNAL
FUNCTION CHECKED_DIV_UNSIGNED : TIME
VAR_INPUT
	IN1 : TIME;
	IN2 : ULINT;
END_VAR
END_FUNCTION

(********************
*
* This operator produces the division of TIME and ANY_NUM.
*
*********************)
FUNCTION DIV_TIME <T: ANY_NUM> : TIME
VAR_INPUT
	IN1 : TIME;
	IN2 : T;
END_VAR
END_FUNCTION

(* Specialized implementation of DIV_TIME for SINT *)
FUNCTION DIV_TIME__SINT : TIME
VAR_INPUT
	IN1 : TIME;
	IN2 : SINT;
END_VAR
	DIV_TIME__SINT := CHECKED_DIV_SIGNED(IN1, IN2);
END_FUNCTION

(* Specialized implementation of DIV_TIME for INT *)
FUNCTION DIV_TIME__INT : TIME
VAR_INPUT
	IN1 : TIME;
	IN2 : INT;
END_VAR
	DIV_TIME__INT := CHECKED_DIV_SIGNED(IN1, IN2);
END_FUNCTION

(* Specialized implementation of DIV_TIME for DINT *)
FUNCTION DIV_TIME__DINT : TIME
VAR_INPUT
	IN1 : TIME;
	IN2 : DINT;
END_VAR
	DIV_TIME__DINT := CHECKED_DIV_SIGNED(IN1, IN2);
END_FUNCTION

(* Specialized implementation of DIV_TIME for LINT *)
FUNCTION DIV_TIME__LINT : TIME
VAR_INPUT
	IN1 : TIME;
	IN2 : LINT;
END_VAR
	DIV_TIME__LINT := CHECKED_DIV_SIGNED(IN1, IN2);
END_FUNCTION

(* Specialized implementation of DIV_TIME for USINT *)
FUNCTION DIV_TIME__USINT : TIME
VAR_INPUT
	IN1 : TIME;
	IN2 : USINT;
END_VAR
	DIV_TIME__USINT := CHECKED_DIV_UNSIGNED(IN1, IN2);
END_FUNCTION

(* Specialized implementation of DIV_TIME for UINT *)
FUNCTION DIV_TIME__UINT : TIME
VAR_INPUT
	IN1 : TIME;
	IN2 : UINT;
END_VAR
	DIV_TIME__UINT := CHECKED_DIV_UNSIGNED(IN1, IN2);
END_FUNCTION

(* Specialized implementation of DIV_TIME for UDINT *)
FUNCTION DIV_TIME__UDINT : TIME
VAR_INPUT
	IN1 : TIME;
	IN2 : UDINT;
END_VAR
	DIV_TIME__UDINT := CHECKED_DIV_UNSIGNED(IN1, IN2);
END_FUNCTION

(* Specialized implementation of DIV_TIME for ULINT *)
FUNCTION DIV_TIME__ULINT : TIME
VAR_INPUT
	IN1 : TIME;
	IN2 : ULINT;
END_VAR
	DIV_TIME__ULINT := CHECKED_DIV_UNSIGNED(IN1, IN2);
END_FUNCTION

(********************
*
* This operator produces the division of LTIME and ANY_NUM.
*
*********************)
FUNCTION DIV_LTIME <T: ANY_NUM> : LTIME
VAR_INPUT
	IN1 : LTIME;
	IN2 : T;
END_VAR
END_FUNCTION

(* Specialized implementation of DIV_LTIME for SINT *)
FUNCTION DIV_LTIME__SINT : LTIME
VAR_INPUT
	IN1 : LTIME;
	IN2 : SINT;
END_VAR
	DIV_LTIME__SINT := CHECKED_DIV_SIGNED(IN1, IN2);
END_FUNCTION

(* Specialized implementation of DIV_LTIME for INT *)
FUNCTION DIV_LTIME__INT : LTIME
VAR_INPUT
	IN1 : LTIME;
	IN2 : INT;
END_VAR
	DIV_LTIME__INT := CHECKED_DIV_SIGNED(IN1, IN2);
END_FUNCTION

(* Specialized implementation of DIV_LTIME for DINT *)
FUNCTION DIV_LTIME__DINT : LTIME
VAR_INPUT
	IN1 : LTIME;
	IN2 : DINT;
END_VAR
	DIV_LTIME__DINT := CHECKED_DIV_SIGNED(IN1, IN2);
END_FUNCTION

(* Specialized implementation of DIV_LTIME for LINT *)
FUNCTION DIV_LTIME__LINT : LTIME
VAR_INPUT
	IN1 : LTIME;
	IN2 : LINT;
END_VAR
	DIV_LTIME__LINT := CHECKED_DIV_SIGNED(IN1, IN2);
END_FUNCTION

(* Specialized implementation of DIV_LTIME for USINT *)
FUNCTION DIV_LTIME__USINT : LTIME
VAR_INPUT
	IN1 : LTIME;
	IN2 : USINT;
END_VAR
	DIV_LTIME__USINT := CHECKED_DIV_UNSIGNED(IN1, IN2);
END_FUNCTION

(* Specialized implementation of DIV_LTIME for UINT *)
FUNCTION DIV_LTIME__UINT : LTIME
VAR_INPUT
	IN1 : LTIME;
	IN2 : UINT;
END_VAR
	DIV_LTIME__UINT := CHECKED_DIV_UNSIGNED(IN1, IN2);
END_FUNCTION

(* Specialized implementation of DIV_LTIME for UDINT *)
FUNCTION DIV_LTIME__UDINT : LTIME
VAR_INPUT
	IN1 : LTIME;
	IN2 : UDINT;
END_VAR
	DIV_LTIME__UDINT := CHECKED_DIV_UNSIGNED(IN1, IN2);
END_FUNCTION

(* Specialized implementation of DIV_LTIME for ULINT *)
FUNCTION DIV_LTIME__ULINT : LTIME
VAR_INPUT
	IN1 : LTIME;
	IN2 : ULINT;
END_VAR
	DIV_LTIME__ULINT := CHECKED_DIV_UNSIGNED(IN1, IN2);
END_FUNCTION

(* Specialized implementation of MUL for TIME and REAL *)
FUNCTION MUL__TIME__REAL : TIME
VAR_INPUT
	IN1 : TIME;
	IN2 : REAL;
END_VAR
	MUL__TIME__REAL := CHECKED_MUL_F32(IN1, IN2);
END_FUNCTION

@EXTERNAL
FUNCTION CHECKED_MUL_F32 : TIME
VAR_INPUT
	IN1 : TIME;
	IN2 : REAL;
END_VAR
END_FUNCTION

(* Specialized implementation of MUL for TIME and LREAL *)
FUNCTION MUL__TIME__LREAL : TIME
VAR_INPUT
	IN1 : TIME;
	IN2 : LREAL;
END_VAR
	MUL__TIME__LREAL := CHECKED_MUL_F64(IN1, IN2);
END_FUNCTION

@EXTERNAL
FUNCTION CHECKED_MUL_F64 : TIME
VAR_INPUT
	IN1 : TIME;
	IN2 : REAL;
END_VAR
END_FUNCTION

(* Specialized implementation of MUL_TIME for REAL *)
FUNCTION MUL_TIME__REAL : TIME
VAR_INPUT
	IN1 : TIME;
	IN2 : REAL;
END_VAR
	MUL_TIME__REAL := CHECKED_MUL_F32(IN1, IN2);
END_FUNCTION

(* Specialized implementation of MUL_TIME for LREAL *)
FUNCTION MUL_TIME__LREAL : TIME
VAR_INPUT
	IN1 : TIME;
	IN2 : LREAL;
END_VAR
	MUL_TIME__LREAL := CHECKED_MUL_F64(IN1, IN2);
END_FUNCTION

(* Specialized implementation of MUL_LTIME for REAL *)
FUNCTION MUL_LTIME__REAL : LTIME
VAR_INPUT
	IN1 : LTIME;
	IN2 : REAL;
END_VAR
	MUL_LTIME__REAL := CHECKED_MUL_F32(IN1, IN2);
END_FUNCTION

(* Specialized implementation of MUL_LTIME for LREAL *)
FUNCTION MUL_LTIME__LREAL : LTIME
VAR_INPUT
	IN1 : LTIME;
	IN2 : LREAL;
END_VAR
	MUL_LTIME__LREAL := CHECKED_MUL_F64(IN1, IN2);
END_FUNCTION

(* Specialized implementation of DIV for TIME and REAL *)
FUNCTION DIV__TIME__REAL : TIME
VAR_INPUT
	IN1 : TIME;
	IN2 : REAL;
END_VAR
	DIV__TIME__REAL := CHECKED_DIV_F32(IN1, IN2);
END_FUNCTION

@EXTERNAL
FUNCTION CHECKED_DIV_F32 : TIME
VAR_INPUT
	IN1 : TIME;
	IN2 : REAL;
END_VAR
END_FUNCTION

(* Specialized implementation of DIV for TIME and LREAL *)
FUNCTION DIV__TIME__LREAL : TIME
VAR_INPUT
	IN1 : TIME;
	IN2 : LREAL;
END_VAR
	DIV__TIME__LREAL := CHECKED_DIV_F64(IN1, IN2);
END_FUNCTION

@EXTERNAL
FUNCTION CHECKED_DIV_F64 : TIME
VAR_INPUT
	IN1 : TIME;
	IN2 : REAL;
END_VAR
END_FUNCTION

(* Specialized implementation of DIV_TIME for REAL *)
FUNCTION DIV_TIME__REAL : TIME
VAR_INPUT
	IN1 : TIME;
	IN2 : REAL;
END_VAR
	DIV_TIME__REAL := CHECKED_DIV_F32(IN1, IN2);
END_FUNCTION

(* Specialized implementation of DIV_TIME for LREAL *)
FUNCTION DIV_TIME__LREAL : TIME
VAR_INPUT
	IN1 : TIME;
	IN2 : LREAL;
END_VAR
	DIV_TIME__LREAL := CHECKED_DIV_F64(IN1, IN2);
END_FUNCTION

(* Specialized implementation of DIV_LTIME for REAL *)
FUNCTION DIV_LTIME__REAL : LTIME
VAR_INPUT
	IN1 : LTIME;
	IN2 : REAL;
END_VAR
	DIV_LTIME__REAL := CHECKED_DIV_F32(IN1, IN2);
END_FUNCTION

(* Specialized implementation of DIV_LTIME for LREAL *)
FUNCTION DIV_LTIME__LREAL : LTIME
VAR_INPUT
	IN1 : LTIME;
	IN2 : LREAL;
END_VAR
	DIV_LTIME__LREAL := CHECKED_DIV_F64(IN1, IN2);
END_FUNCTION

(* ---- endianness_conversion_functions.st ---- *)
// ANY_REAL and ANY_BIT bit-width constraint >=16 -> how?

(********************
*
* Converts little endian data format to big endian data format
*
*********************)
{external}
FUNCTION TO_BIG_ENDIAN<T: ANY> : T
VAR_INPUT
	in : T;
END_VAR
END_FUNCTION

(********************
*
* Converts big endian data format to little endian data format
*
*********************)
{external}
FUNCTION TO_LITTLE_ENDIAN<T: ANY> : T
VAR_INPUT
	in : T;
END_VAR
END_FUNCTION

(********************
*
* Converts to little endian data format from big endian data format
*
*********************)
{external}
FUNCTION FROM_BIG_ENDIAN<T: ANY> : T
VAR_INPUT
	in : T;
END_VAR
END_FUNCTION

(********************
*
* Converts to big endian data format from little endian data format
*
*********************)
{external}
FUNCTION FROM_LITTLE_ENDIAN<T: ANY> : T
VAR_INPUT
	in : T;
END_VAR
END_FUNCTION

(* ---- extra_functions.st ---- *)
(******************************************************************************
*
* Converts BYTE to STRING.
*
******************************************************************************)
FUNCTION BYTE_TO_STRING : STRING[__STRING_LENGTH]
VAR_INPUT
    IN: BYTE;
END_VAR
    BYTE_TO_STRING_EXT(IN, BYTE_TO_STRING);
END_FUNCTION

{external}
FUNCTION BYTE_TO_STRING_EXT : DINT
VAR_INPUT
    IN: BYTE;
END_VAR
VAR_IN_OUT
    OUT: STRING[__STRING_LENGTH];
END_VAR
END_FUNCTION

{external}
FUNCTION LWORD_TO_STRING_EXT : DINT
VAR_INPUT
    IN: LWORD;
END_VAR
VAR_IN_OUT
    OUT: STRING[__STRING_LENGTH];
END_VAR
END_FUNCTION

(******************************************************************************
*
* Converts LWORD to STRING.
*
******************************************************************************)
FUNCTION LWORD_TO_STRING : STRING[__STRING_LENGTH]
VAR_INPUT
    IN: LWORD;
END_VAR
    LWORD_TO_STRING_EXT(IN, LWORD_TO_STRING);
END_FUNCTION

(******************************************************************************
*
* Converts DWORD to STRING.
*
******************************************************************************)
FUNCTION DWORD_TO_STRING : STRING[__STRING_LENGTH]
VAR_INPUT
    IN: DWORD;
END_VAR
    LWORD_TO_STRING_EXT(IN, DWORD_TO_STRING);
END_FUNCTION

{external}
FUNCTION LINT_TO_STRING_EXT : DINT
VAR_INPUT
    IN: LINT;
END_VAR
VAR_IN_OUT
    OUT: STRING[__STRING_LENGTH];
END_VAR
END_FUNCTION

(******************************************************************************
*
* Converts LINT to STRING.
*
******************************************************************************)
FUNCTION LINT_TO_STRING : STRING[__STRING_LENGTH]
VAR_INPUT
    IN: LINT;
END_VAR
    LINT_TO_STRING_EXT(IN, LINT_TO_STRING);
END_FUNCTION

(******************************************************************************
*
* Converts DINT to STRING.
*
******************************************************************************)
FUNCTION DINT_TO_STRING : STRING[__STRING_LENGTH]
VAR_INPUT
    IN: DINT;
END_VAR
    LINT_TO_STRING_EXT(IN, DINT_TO_STRING);
END_FUNCTION

{external}
FUNCTION LREAL_TO_STRING_EXT : DINT
VAR_INPUT
    IN: LREAL;
END_VAR
VAR_IN_OUT
    OUT: STRING[__STRING_LENGTH];
END_VAR
END_FUNCTION

(******************************************************************************
*
* Converts BYTE to WSTRING.
*
******************************************************************************)
FUNCTION BYTE_TO_WSTRING : WSTRING[__STRING_LENGTH]
VAR_INPUT
    IN: BYTE;
END_VAR
    STRING_TO_WSTRING_EXT(BYTE_TO_STRING(IN), BYTE_TO_WSTRING);
END_FUNCTION

(******************************************************************************
*
* Converts LWORD to WSTRING.
*
******************************************************************************)
FUNCTION LWORD_TO_WSTRING : WSTRING[__STRING_LENGTH]
VAR_INPUT
    IN: LWORD;
END_VAR
    STRING_TO_WSTRING_EXT(LWORD_TO_STRING(IN), LWORD_TO_WSTRING);
END_FUNCTION

(******************************************************************************
*
* Converts DWORD to WSTRING.
*
******************************************************************************)
FUNCTION DWORD_TO_WSTRING : WSTRING[__STRING_LENGTH]
VAR_INPUT
    IN: DWORD;
END_VAR
    DWORD_TO_WSTRING := LWORD_TO_WSTRING(IN);
END_FUNCTION

(******************************************************************************
*
* Converts LINT to WSTRING.
*
******************************************************************************)
FUNCTION LINT_TO_WSTRING : WSTRING[__STRING_LENGTH]
VAR_INPUT
    IN: LINT;
END_VAR
    STRING_TO_WSTRING_EXT(LINT_TO_STRING(IN), LINT_TO_WSTRING);
END_FUNCTION

(******************************************************************************
*
* Converts DINT to WSTRING.
*
******************************************************************************)
FUNCTION DINT_TO_WSTRING : WSTRING[__STRING_LENGTH]
VAR_INPUT
    IN: DINT;
END_VAR
    DINT_TO_WSTRING := LINT_TO_WSTRING(IN);
END_FUNCTION

(******************************************************************************
*
* Converts LREAL to STRING.
*
******************************************************************************)
FUNCTION LREAL_TO_STRING : STRING[__STRING_LENGTH]
VAR_INPUT
    IN: LREAL;
END_VAR
    LREAL_TO_STRING_EXT(IN, LREAL_TO_STRING);
END_FUNCTION

(******************************************************************************
*
* Converts REAL to STRING.
*
******************************************************************************)
FUNCTION REAL_TO_STRING : STRING[__STRING_LENGTH]
VAR_INPUT
    IN: REAL;
END_VAR
    LREAL_TO_STRING_EXT(IN, REAL_TO_STRING);
END_FUNCTION

(******************************************************************************
*
* Converts LREAL to WSTRING.
*
******************************************************************************)
FUNCTION LREAL_TO_WSTRING : WSTRING[__STRING_LENGTH]
VAR_INPUT
    IN: LREAL;
END_VAR
    STRING_TO_WSTRING_EXT(LREAL_TO_STRING(IN), LREAL_TO_WSTRING);
END_FUNCTION

(******************************************************************************
*
* Converts REAL to WSTRING.
*
******************************************************************************)
FUNCTION REAL_TO_WSTRING : WSTRING[__STRING_LENGTH]
VAR_INPUT
    IN: REAL;
END_VAR
    REAL_TO_WSTRING := LREAL_TO_WSTRING(IN);
END_FUNCTION

(******************************************************************************
*
* Converts TOD to LWORD.
*
******************************************************************************)
FUNCTION TOD_TO_LWORD : LWORD
VAR_INPUT
    IN: TOD;
END_VAR
    TOD_TO_LWORD := IN;
END_FUNCTION

(******************************************************************************
*
* Converts DT to LWORD.
*
******************************************************************************)
FUNCTION DT_TO_LWORD : LWORD
VAR_INPUT
    IN: TOD;
END_VAR
    DT_TO_LWORD := IN;
END_FUNCTION

(******************************************************************************
*
* Converts DATE to LWORD.
*
******************************************************************************)
FUNCTION DATE_TO_LWORD : LWORD
VAR_INPUT
    IN: DATE;
END_VAR
    DATE_TO_LWORD := IN;
END_FUNCTION

(******************************************************************************
*
* Converts TIME to LWORD.
*
******************************************************************************)
FUNCTION TIME_TO_LWORD : LWORD
VAR_INPUT
    IN: TIME;
END_VAR
    TIME_TO_LWORD := IN;
END_FUNCTION

(******************************************************************************
*
* Converts STRING to LINT.
*
******************************************************************************)
{external}
FUNCTION STRING_TO_LINT : LINT
VAR_INPUT {ref}
    IN: STRING;
END_VAR
END_FUNCTION

(******************************************************************************
*
* Converts WSTRING to LINT.
*
******************************************************************************)
FUNCTION WSTRING_TO_LINT : LINT
VAR_INPUT {ref}
    IN: WSTRING;
END_VAR
VAR_TEMP
    STR: STRING;
END_VAR
    WSTRING_TO_STRING_EXT(IN, STR);
    WSTRING_TO_LINT := STRING_TO_LINT(STR);
END_FUNCTION

(******************************************************************************
*
* Converts TIME to LINT.
*
******************************************************************************)
FUNCTION TIME_TO_LINT : LINT
VAR_INPUT
    IN: TIME;
END_VAR
    TIME_TO_LINT := IN;
END_FUNCTION

FUNCTION TOD_TO_LINT : LINT
VAR_INPUT
    IN: TOD;
END_VAR
    TOD_TO_LINT := IN;
END_FUNCTION

(******************************************************************************
*
* Converts DT to LINT.
*
******************************************************************************)
FUNCTION DT_TO_LINT : LINT
VAR_INPUT
    IN: DT;
END_VAR
    DT_TO_LINT := IN;
END_FUNCTION

(******************************************************************************
*
* Converts DT to ULINT.
*
******************************************************************************)
FUNCTION DT_TO_ULINT : ULINT
VAR_INPUT
    IN: DT;
END_VAR
    DT_TO_ULINT := IN;
END_FUNCTION

(******************************************************************************
*
* Converts TIME to ULINT.
*
******************************************************************************)
FUNCTION TIME_TO_ULINT : ULINT
VAR_INPUT
    IN: DT;
END_VAR
    TIME_TO_ULINT := IN;
END_FUNCTION

(******************************************************************************
*
* Converts DATE to ULINT.
*
******************************************************************************)
FUNCTION DATE_TO_ULINT : ULINT
VAR_INPUT
    IN: DATE;
END_VAR
    DATE_TO_ULINT := IN;
END_FUNCTION

(******************************************************************************
*
* Converts TOD to ULINT.
*
******************************************************************************)
FUNCTION TOD_TO_ULINT : ULINT
VAR_INPUT
    IN: TOD;
END_VAR
    TOD_TO_ULINT := IN;
END_FUNCTION

(******************************************************************************
*
* Converts STRING to DINT.
*
******************************************************************************)
{external}
FUNCTION STRING_TO_DINT : DINT
VAR_INPUT {ref}
    IN: STRING;
END_VAR
END_FUNCTION

(******************************************************************************
*
* Converts WSTRING to DINT.
*
******************************************************************************)
FUNCTION WSTRING_TO_DINT : DINT
VAR_INPUT {ref}
    IN: WSTRING;
END_VAR
VAR_TEMP
    STR: STRING;
END_VAR
    WSTRING_TO_STRING_EXT(IN, STR);
    WSTRING_TO_DINT := STRING_TO_LINT(STR);
END_FUNCTION

(******************************************************************************
*
* Converts STRING to LREAL.
*
******************************************************************************)
{external}
FUNCTION STRING_TO_LREAL : LREAL
VAR_INPUT {ref}
    IN: STRING;
END_VAR
END_FUNCTION

(******************************************************************************
*
* Converts STRING to REAL.
*
******************************************************************************)
{external}
FUNCTION STRING_TO_REAL : REAL
VAR_INPUT {ref}
    IN: STRING;
END_VAR
END_FUNCTION

(******************************************************************************
*
* Converts WSTRING to LREAL.
*
******************************************************************************)
FUNCTION WSTRING_TO_LREAL : LREAL
VAR_INPUT {ref}
    IN: WSTRING;
END_VAR
VAR_TEMP
    STR: STRING;
END_VAR
    WSTRING_TO_STRING_EXT(IN, STR);
    WSTRING_TO_LREAL := STRING_TO_LREAL(STR);
END_FUNCTION

(******************************************************************************
*
* Converts WSTRING to REAL.
*
******************************************************************************)
FUNCTION WSTRING_TO_REAL : REAL
VAR_INPUT {ref}
    IN: WSTRING;
END_VAR
VAR_TEMP
    STR: STRING;
END_VAR
    WSTRING_TO_STRING_EXT(IN, STR);
    WSTRING_TO_REAL := STRING_TO_REAL(STR);
END_FUNCTION

(******************************************************************************
*
* Converts TIME to LREAL.
*
******************************************************************************)
FUNCTION TIME_TO_LREAL : LREAL
VAR_INPUT
    IN: TIME;
END_VAR
    TIME_TO_LREAL := IN;
END_FUNCTION

(******************************************************************************
*
* Converts LWORD to TIME.
*
******************************************************************************)
FUNCTION LWORD_TO_TIME : TIME
VAR_INPUT
    IN: LWORD;
END_VAR
    LWORD_TO_TIME := IN;
END_FUNCTION

(******************************************************************************
*
* Converts LREAL to TIME.
*
******************************************************************************)
FUNCTION LREAL_TO_TIME : TIME
VAR_INPUT
    IN: LREAL;
END_VAR
// seconds.millis? round as nanos?
    LREAL_TO_TIME := ROUND(IN);
END_FUNCTION

(******************************************************************************
*
* Converts LINT to TIME.
*
******************************************************************************)
FUNCTION LINT_TO_TIME : TIME
VAR_INPUT
    IN: LINT;
END_VAR
    LINT_TO_TIME := IN;
END_FUNCTION

(******************************************************************************
*
* Converts LWORD to DATE.
*
******************************************************************************)
FUNCTION LWORD_TO_DATE : DATE
VAR_INPUT
    IN: LWORD;
END_VAR
    LWORD_TO_DATE := IN;
END_FUNCTION

(******************************************************************************
*
* Converts ULINT to DATE.
*
******************************************************************************)
FUNCTION ULINT_TO_DATE : DATE
VAR_INPUT
    IN: ULINT;
END_VAR
    ULINT_TO_DATE := IN;
END_FUNCTION

(******************************************************************************
*
* Converts ULINT to DT.
*
******************************************************************************)
FUNCTION ULINT_TO_DT : DT
VAR_INPUT
    IN: ULINT;
END_VAR
    ULINT_TO_DT := IN;
END_FUNCTION

(******************************************************************************
*
* Converts LWORD to DT.
*
******************************************************************************)
FUNCTION LWORD_TO_DT : DT
VAR_INPUT
    IN: LWORD;
END_VAR
    LWORD_TO_DT := IN;
END_FUNCTION

(******************************************************************************
*
* Converts LWORD to TOD.
*
******************************************************************************)
FUNCTION LWORD_TO_TOD : TOD
VAR_INPUT
    IN: LWORD;
END_VAR
    LWORD_TO_TOD := IN;
END_FUNCTION

(******************************************************************************
*
* Converts LINT to TOD.
*
******************************************************************************)
FUNCTION LINT_TO_TOD : TOD
VAR_INPUT
    IN: LINT;
END_VAR
    LINT_TO_TOD := IN;
END_FUNCTION

(******************************************************************************
*
* Converts LINT to BOOL.
*
******************************************************************************)
FUNCTION LINT_TO_BOOL : BOOL
VAR_INPUT
    IN: LINT;
END_VAR
   IF IN = 0 THEN
    LINT_TO_BOOL := FALSE;
   ELSE
    LINT_TO_BOOL := TRUE;
   END_IF;
END_FUNCTION

(******************************************************************************
*
* Converts DINT to BOOL.
*
******************************************************************************)
FUNCTION DINT_TO_BOOL : BOOL
VAR_INPUT
    IN: DINT;
END_VAR
   DINT_TO_BOOL := LINT_TO_BOOL(IN);
END_FUNCTION

(******************************************************************************
*
* Truncate REAL_TYPE to INT_TYPE.
*
******************************************************************************)
FUNCTION TRUNC<T: ANY_REAL> : LINT
VAR_INPUT
    IN: T;
END_VAR
END_FUNCTION

FUNCTION TRUNC__REAL : LINT
VAR_INPUT
    IN: REAL;
END_VAR
    TRUNC__REAL := IN;
END_FUNCTION

FUNCTION TRUNC__LREAL : LINT
VAR_INPUT
    IN: LREAL;
END_VAR
    TRUNC__LREAL := IN;
END_FUNCTION

(******************************************************************************
*
* Returns the local TIME since midnight, which can be used make relative measurements
* by calculating the difference between TIME return-values.
*
******************************************************************************)
{external}
FUNCTION TIME : TIME END_FUNCTION

(* ---- num.st ---- *)
/* (************************** */
/*  * */
/*  *This operator returns the absolute value of a number. */
/*  * */
/* *************************) */
/* FUNCTION ABS<T : ANY_NUM> : T */
/* VAR_INPUT */
/* 	IN : T; */
/* END_VAR */

/* END_FUNCTION */

(* Specialized implementation of ABS for DINT *)
/* FUNCTION ABS__DINT : DINT */
FUNCTION ABS : DINT //__DINT : DINT
VAR_INPUT
	IN : DINT;
END_VAR
	ABS := IN;
	/* ABS__DINT := IN; */
	IF ABS < 0 THEN
	/* IF ABS__DINT < 0 THEN */
		ABS := -1 * ABS;
		/* ABS__DINT := -1 * ABS__DINT; */
	END_IF
END_FUNCTION

/* (* Specialized implementation of ABS for LINT *) */
/* FUNCTION ABS__LINT : LINT */
/* VAR_INPUT */
/* 	IN : LINT; */
/* END_VAR */
/* 	ABS__LINT := IN; */
/* 	IF ABS__LINT < 0 THEN */
/* 		ABS__LINT := -1 * ABS__LINT; */
/* 	END_IF */
/* END_FUNCTION */

(* ---- num_conversion.st ---- *)
(**************************
 *
 * Rounds a given ANY_REAL to the nearest integer
 * Rounds half values away from zero
 *
*************************)
{external}
FUNCTION ROUND<T : ANY_REAL> : T
VAR_INPUT
	in : T;
END_VAR
END_FUNCTION

(********************
*
* Converts LREAL to REAL
*
*********************)
FUNCTION LREAL_TO_REAL : REAL
VAR_INPUT
	in : LREAL;
END_VAR
	LREAL_TO_REAL := in;
END_FUNCTION

(********************
*
* Converts LREAL to LINT
*
*********************)
FUNCTION LREAL_TO_LINT : LINT
VAR_INPUT
	in : LREAL;
END_VAR
	LREAL_TO_LINT := ROUND(in);
END_FUNCTION

(********************
*
* Converts LREAL to DINT
*
*********************)
FUNCTION LREAL_TO_DINT : DINT
VAR_INPUT
	in : LREAL;
END_VAR
	LREAL_TO_DINT := ROUND(in);
END_FUNCTION

(********************
*
* Converts LREAL to INT
*
*********************)
FUNCTION LREAL_TO_INT : INT
VAR_INPUT
	in : LREAL;
END_VAR
	LREAL_TO_INT := ROUND(in);
END_FUNCTION

(********************
*
* Converts LREAL to SINT
*
*********************)
FUNCTION LREAL_TO_SINT : SINT
VAR_INPUT
	in : LREAL;
END_VAR
	LREAL_TO_SINT := ROUND(in);
END_FUNCTION

(********************
*
* Converts LREAL to ULINT
*
*********************)
FUNCTION LREAL_TO_ULINT : ULINT
VAR_INPUT
	in : LREAL;
END_VAR
	LREAL_TO_ULINT := ROUND(in);
END_FUNCTION

(********************
*
* Converts LREAL to UDINT
*
*********************)
FUNCTION LREAL_TO_UDINT : UDINT
VAR_INPUT
	in : LREAL;
END_VAR
	LREAL_TO_UDINT := ROUND(in);
END_FUNCTION

(********************
*
* Converts LREAL to UINT
*
*********************)
FUNCTION LREAL_TO_UINT : UINT
VAR_INPUT
	in : LREAL;
END_VAR
	LREAL_TO_UINT := ROUND(in);
END_FUNCTION

(********************
*
* Converts LREAL to USINT
*
*********************)
FUNCTION LREAL_TO_USINT : USINT
VAR_INPUT
	in : LREAL;
END_VAR
	LREAL_TO_USINT := ROUND(in);
END_FUNCTION

(********************
*
* Converts REAL to LREAL
*
*********************)
FUNCTION REAL_TO_LREAL : LREAL
VAR_INPUT
	in : REAL;
END_VAR
	REAL_TO_LREAL := in;
END_FUNCTION

(********************
*
* Converts REAL to LINT
*
*********************)
FUNCTION REAL_TO_LINT : LINT
VAR_INPUT
	in : REAL;
END_VAR
	REAL_TO_LINT := ROUND(in);
END_FUNCTION

(********************
*
* Converts REAL to DINT
*
*********************)
FUNCTION REAL_TO_DINT : DINT
VAR_INPUT
	in : REAL;
END_VAR
	REAL_TO_DINT := ROUND(in);
END_FUNCTION

(********************
*
* Converts REAL to INT
*
*********************)
FUNCTION REAL_TO_INT : INT
VAR_INPUT
	in : REAL;
END_VAR
	REAL_TO_INT := ROUND(in);
END_FUNCTION

(********************
*
* Converts REAL to SINT
*
*********************)
FUNCTION REAL_TO_SINT : SINT
VAR_INPUT
	in : REAL;
END_VAR
	REAL_TO_SINT := ROUND(in);
END_FUNCTION

(********************
*
* Converts REAL to ULINT
*
*********************)
FUNCTION REAL_TO_ULINT : ULINT
VAR_INPUT
	in : REAL;
END_VAR
	REAL_TO_ULINT := ROUND(in);
END_FUNCTION

(********************
*
* Converts REAL to UDINT
*
*********************)
FUNCTION REAL_TO_UDINT : UDINT
VAR_INPUT
	in : REAL;
END_VAR
	REAL_TO_UDINT := ROUND(in);
END_FUNCTION

(********************
*
* Converts REAL to UINT
*
*********************)
FUNCTION REAL_TO_UINT : UINT
VAR_INPUT
	in : REAL;
END_VAR
	REAL_TO_UINT := ROUND(in);
END_FUNCTION

(********************
*
* Converts REAL to USINT
*
*********************)
FUNCTION REAL_TO_USINT : USINT
VAR_INPUT
	in : REAL;
END_VAR
	REAL_TO_USINT := ROUND(in);
END_FUNCTION

(********************
*
* Converts LINT to LREAL
*
*********************)
FUNCTION LINT_TO_LREAL : LREAL
VAR_INPUT
	in : LINT;
END_VAR
	LINT_TO_LREAL := in;
END_FUNCTION

(********************
*
* Converts LINT to REAL
*
*********************)
FUNCTION LINT_TO_REAL : REAL
VAR_INPUT
	in : LINT;
END_VAR
	LINT_TO_REAL := in;
END_FUNCTION

(********************
*
* Converts LINT to DINT
*
*********************)
FUNCTION LINT_TO_DINT : DINT
VAR_INPUT
	in : LINT;
END_VAR
	LINT_TO_DINT := in;
END_FUNCTION

(********************
*
* Converts LINT to INT
*
*********************)
FUNCTION LINT_TO_INT : INT
VAR_INPUT
	in : LINT;
END_VAR
	LINT_TO_INT := in;
END_FUNCTION

(********************
*
* Converts LINT to SINT
*
*********************)
FUNCTION LINT_TO_SINT : SINT
VAR_INPUT
	in : LINT;
END_VAR
	LINT_TO_SINT := in;
END_FUNCTION

(********************
*
* Converts LINT to ULINT
*
*********************)
FUNCTION LINT_TO_ULINT : ULINT
VAR_INPUT
	in : LINT;
END_VAR
	LINT_TO_ULINT := in;
END_FUNCTION

(********************
*
* Converts LINT to UDINT
*
*********************)
FUNCTION LINT_TO_UDINT : UDINT
VAR_INPUT
	in : LINT;
END_VAR
	LINT_TO_UDINT := in;
END_FUNCTION

(********************
*
* Converts LINT to UINT
*
*********************)
FUNCTION LINT_TO_UINT : UINT
VAR_INPUT
	in : LINT;
END_VAR
	LINT_TO_UINT := in;
END_FUNCTION

(********************
*
* Converts LINT to USINT
*
*********************)
FUNCTION LINT_TO_USINT : USINT
VAR_INPUT
	in : LINT;
END_VAR
	LINT_TO_USINT := in;
END_FUNCTION

(********************
*
* Converts DINT to LREAL
*
*********************)
FUNCTION DINT_TO_LREAL : LREAL
VAR_INPUT
	in : DINT;
END_VAR
	DINT_TO_LREAL := in;
END_FUNCTION

(********************
*
* Converts DINT to REAL
*
*********************)
FUNCTION DINT_TO_REAL : REAL
VAR_INPUT
	in : DINT;
END_VAR
	DINT_TO_REAL := in;
END_FUNCTION

(********************
*
* Converts DINT to LINT
*
*********************)
FUNCTION DINT_TO_LINT : LINT
VAR_INPUT
	in : DINT;
END_VAR
	DINT_TO_LINT := in;
END_FUNCTION

(********************
*
* Converts DINT to INT
*
*********************)
FUNCTION DINT_TO_INT : INT
VAR_INPUT
	in : DINT;
END_VAR
	DINT_TO_INT := in;
END_FUNCTION

(********************
*
* Converts DINT to SINT
*
*********************)
FUNCTION DINT_TO_SINT : SINT
VAR_INPUT
	in : DINT;
END_VAR
	DINT_TO_SINT := in;
END_FUNCTION

(********************
*
* Converts DINT to ULINT
*
*********************)
FUNCTION DINT_TO_ULINT : ULINT
VAR_INPUT
	in : DINT;
END_VAR
	DINT_TO_ULINT := in;
END_FUNCTION

(********************
*
* Converts DINT to UDINT
*
*********************)
FUNCTION DINT_TO_UDINT : UDINT
VAR_INPUT
	in : DINT;
END_VAR
	DINT_TO_UDINT := in;
END_FUNCTION

(********************
*
* Converts DINT to UINT
*
*********************)
FUNCTION DINT_TO_UINT : UINT
VAR_INPUT
	in : DINT;
END_VAR
	DINT_TO_UINT := in;
END_FUNCTION

(********************
*
* Converts DINT to USINT
*
*********************)
FUNCTION DINT_TO_USINT : USINT
VAR_INPUT
	in : DINT;
END_VAR
	DINT_TO_USINT := in;
END_FUNCTION

(********************
*
* Converts INT to LREAL
*
*********************)
FUNCTION INT_TO_LREAL : LREAL
VAR_INPUT
	in : INT;
END_VAR
	INT_TO_LREAL := in;
END_FUNCTION

(********************
*
* Converts INT to REAL
*
*********************)
FUNCTION INT_TO_REAL : REAL
VAR_INPUT
	in : INT;
END_VAR
	INT_TO_REAL := in;
END_FUNCTION

(********************
*
* Converts INT to LINT
*
*********************)
FUNCTION INT_TO_LINT : LINT
VAR_INPUT
	in : INT;
END_VAR
	INT_TO_LINT := in;
END_FUNCTION

(********************
*
* Converts INT to DINT
*
*********************)
FUNCTION INT_TO_DINT : DINT
VAR_INPUT
	in : INT;
END_VAR
	INT_TO_DINT := in;
END_FUNCTION

(********************
*
* Converts INT to SINT
*
*********************)
FUNCTION INT_TO_SINT : SINT
VAR_INPUT
	in : INT;
END_VAR
	INT_TO_SINT := in;
END_FUNCTION

(********************
*
* Converts INT to ULINT
*
*********************)
FUNCTION INT_TO_ULINT : ULINT
VAR_INPUT
	in : INT;
END_VAR
	INT_TO_ULINT := in;
END_FUNCTION

(********************
*
* Converts INT to UDINT
*
*********************)
FUNCTION INT_TO_UDINT : UDINT
VAR_INPUT
	in : INT;
END_VAR
	INT_TO_UDINT := in;
END_FUNCTION

(********************
*
* Converts INT to UINT
*
*********************)
FUNCTION INT_TO_UINT : UINT
VAR_INPUT
	in : INT;
END_VAR
	INT_TO_UINT := in;
END_FUNCTION

(********************
*
* Converts INT to USINT
*
*********************)
FUNCTION INT_TO_USINT : USINT
VAR_INPUT
	in : INT;
END_VAR
	INT_TO_USINT := in;
END_FUNCTION

(********************
*
* Converts SINT to LREAL
*
*********************)
FUNCTION SINT_TO_LREAL : LREAL
VAR_INPUT
	in : SINT;
END_VAR
	SINT_TO_LREAL := in;
END_FUNCTION

(********************
*
* Converts SINT to REAL
*
*********************)
FUNCTION SINT_TO_REAL : REAL
VAR_INPUT
	in : SINT;
END_VAR
	SINT_TO_REAL := in;
END_FUNCTION

(********************
*
* Converts SINT to LINT
*
*********************)
FUNCTION SINT_TO_LINT : LINT
VAR_INPUT
	in : SINT;
END_VAR
	SINT_TO_LINT := in;
END_FUNCTION

(********************
*
* Converts SINT to DINT
*
*********************)
FUNCTION SINT_TO_DINT : DINT
VAR_INPUT
	in : SINT;
END_VAR
	SINT_TO_DINT := in;
END_FUNCTION

(********************
*
* Converts SINT to INT
*
*********************)
FUNCTION SINT_TO_INT : INT
VAR_INPUT
	in : SINT;
END_VAR
	SINT_TO_INT := in;
END_FUNCTION

(********************
*
* Converts SINT to ULINT
*
*********************)
FUNCTION SINT_TO_ULINT : ULINT
VAR_INPUT
	in : SINT;
END_VAR
	SINT_TO_ULINT := in;
END_FUNCTION

(********************
*
* Converts SINT to UDINT
*
*********************)
FUNCTION SINT_TO_UDINT : UDINT
VAR_INPUT
	in : SINT;
END_VAR
	SINT_TO_UDINT := in;
END_FUNCTION

(********************
*
* Converts SINT to UINT
*
*********************)
FUNCTION SINT_TO_UINT : UINT
VAR_INPUT
	in : SINT;
END_VAR
	SINT_TO_UINT := in;
END_FUNCTION

(********************
*
* Converts SINT to USINT
*
*********************)
FUNCTION SINT_TO_USINT : USINT
VAR_INPUT
	in : SINT;
END_VAR
	SINT_TO_USINT := in;
END_FUNCTION

(********************
*
* Converts ULINT to LREAL
*
*********************)
FUNCTION ULINT_TO_LREAL : LREAL
VAR_INPUT
	in : ULINT;
END_VAR
	ULINT_TO_LREAL := in;
END_FUNCTION

(********************
*
* Converts ULINT to REAL
*
*********************)
FUNCTION ULINT_TO_REAL : REAL
VAR_INPUT
	in : ULINT;
END_VAR
	ULINT_TO_REAL := in;
END_FUNCTION

(********************
*
* Converts ULINT to LINT
*
*********************)
FUNCTION ULINT_TO_LINT : LINT
VAR_INPUT
	in : ULINT;
END_VAR
	ULINT_TO_LINT := in;
END_FUNCTION

(********************
*
* Converts ULINT to DINT
*
*********************)
FUNCTION ULINT_TO_DINT : DINT
VAR_INPUT
	in : ULINT;
END_VAR
	ULINT_TO_DINT := in;
END_FUNCTION

(********************
*
* Converts ULINT to INT
*
*********************)
FUNCTION ULINT_TO_INT : INT
VAR_INPUT
	in : ULINT;
END_VAR
	ULINT_TO_INT := in;
END_FUNCTION

(********************
*
* Converts ULINT to SINT
*
*********************)
FUNCTION ULINT_TO_SINT : SINT
VAR_INPUT
	in : ULINT;
END_VAR
	ULINT_TO_SINT := in;
END_FUNCTION

(********************
*
* Converts ULINT to UDINT
*
*********************)
FUNCTION ULINT_TO_UDINT : UDINT
VAR_INPUT
	in : ULINT;
END_VAR
	ULINT_TO_UDINT := in;
END_FUNCTION

(********************
*
* Converts ULINT to UINT
*
*********************)
FUNCTION ULINT_TO_UINT : UINT
VAR_INPUT
	in : ULINT;
END_VAR
	ULINT_TO_UINT := in;
END_FUNCTION

(********************
*
* Converts ULINT to USINT
*
*********************)
FUNCTION ULINT_TO_USINT : USINT
VAR_INPUT
	in : ULINT;
END_VAR
	ULINT_TO_USINT := in;
END_FUNCTION

(********************
*
* Converts UDINT to LREAL
*
*********************)
FUNCTION UDINT_TO_LREAL : LREAL
VAR_INPUT
	in : UDINT;
END_VAR
	UDINT_TO_LREAL := in;
END_FUNCTION

(********************
*
* Converts UDINT to REAL
*
*********************)
FUNCTION UDINT_TO_REAL : REAL
VAR_INPUT
	in : UDINT;
END_VAR
	UDINT_TO_REAL := in;
END_FUNCTION

(********************
*
* Converts UDINT to LINT
*
*********************)
FUNCTION UDINT_TO_LINT : LINT
VAR_INPUT
	in : UDINT;
END_VAR
	UDINT_TO_LINT := in;
END_FUNCTION

(********************
*
* Converts UDINT to DINT
*
*********************)
FUNCTION UDINT_TO_DINT : DINT
VAR_INPUT
	in : UDINT;
END_VAR
	UDINT_TO_DINT := in;
END_FUNCTION

(********************
*
* Converts UDINT to INT
*
*********************)
FUNCTION UDINT_TO_INT : INT
VAR_INPUT
	in : UDINT;
END_VAR
	UDINT_TO_INT := in;
END_FUNCTION

(********************
*
* Converts UDINT to SINT
*
*********************)
FUNCTION UDINT_TO_SINT : SINT
VAR_INPUT
	in : UDINT;
END_VAR
	UDINT_TO_SINT := in;
END_FUNCTION

(********************
*
* Converts UDINT to ULINT
*
*********************)
FUNCTION UDINT_TO_ULINT : ULINT
VAR_INPUT
	in : UDINT;
END_VAR
	UDINT_TO_ULINT := in;
END_FUNCTION

(********************
*
* Converts UDINT to UINT
*
*********************)
FUNCTION UDINT_TO_UINT : UINT
VAR_INPUT
	in : UDINT;
END_VAR
	UDINT_TO_UINT := in;
END_FUNCTION

(********************
*
* Converts UDINT to USINT
*
*********************)
FUNCTION UDINT_TO_USINT : USINT
VAR_INPUT
	in : UDINT;
END_VAR
	UDINT_TO_USINT := in;
END_FUNCTION

(********************
*
* Converts UINT to LREAL
*
*********************)
FUNCTION UINT_TO_LREAL : LREAL
VAR_INPUT
	in : UINT;
END_VAR
	UINT_TO_LREAL := in;
END_FUNCTION

(********************
*
* Converts UINT to REAL
*
*********************)
FUNCTION UINT_TO_REAL : REAL
VAR_INPUT
	in : UINT;
END_VAR
	UINT_TO_REAL := in;
END_FUNCTION

(********************
*
* Converts UINT to LINT
*
*********************)
FUNCTION UINT_TO_LINT : LINT
VAR_INPUT
	in : UINT;
END_VAR
	UINT_TO_LINT := in;
END_FUNCTION

(********************
*
* Converts UINT to DINT
*
*********************)
FUNCTION UINT_TO_DINT : DINT
VAR_INPUT
	in : UINT;
END_VAR
	UINT_TO_DINT := in;
END_FUNCTION

(********************
*
* Converts UINT to INT
*
*********************)
FUNCTION UINT_TO_INT : INT
VAR_INPUT
	in : UINT;
END_VAR
	UINT_TO_INT := in;
END_FUNCTION

(********************
*
* Converts UINT to SINT
*
*********************)
FUNCTION UINT_TO_SINT : SINT
VAR_INPUT
	in : UINT;
END_VAR
	UINT_TO_SINT := in;
END_FUNCTION

(********************
*
* Converts UINT to ULINT
*
*********************)
FUNCTION UINT_TO_ULINT : ULINT
VAR_INPUT
	in : UINT;
END_VAR
	UINT_TO_ULINT := in;
END_FUNCTION

(********************
*
* Converts UINT to UDINT
*
*********************)
FUNCTION UINT_TO_UDINT : UDINT
VAR_INPUT
	in : UINT;
END_VAR
	UINT_TO_UDINT := in;
END_FUNCTION

(********************
*
* Converts UINT to USINT
*
*********************)
FUNCTION UINT_TO_USINT : USINT
VAR_INPUT
	in : UINT;
END_VAR
	UINT_TO_USINT := in;
END_FUNCTION

(********************
*
* Converts USINT to LREAL
*
*********************)
FUNCTION USINT_TO_LREAL : LREAL
VAR_INPUT
	in : USINT;
END_VAR
	USINT_TO_LREAL := in;
END_FUNCTION

(********************
*
* Converts USINT to REAL
*
*********************)
FUNCTION USINT_TO_REAL : REAL
VAR_INPUT
	in : USINT;
END_VAR
	USINT_TO_REAL := in;
END_FUNCTION

(********************
*
* Converts USINT to LINT
*
*********************)
FUNCTION USINT_TO_LINT : LINT
VAR_INPUT
	in : USINT;
END_VAR
	USINT_TO_LINT := in;
END_FUNCTION

(********************
*
* Converts USINT to DINT
*
*********************)
FUNCTION USINT_TO_DINT : DINT
VAR_INPUT
	in : USINT;
END_VAR
	USINT_TO_DINT := in;
END_FUNCTION

(********************
*
* Converts USINT to INT
*
*********************)
FUNCTION USINT_TO_INT : INT
VAR_INPUT
	in : USINT;
END_VAR
	USINT_TO_INT := in;
END_FUNCTION

(********************
*
* Converts USINT to SINT
*
*********************)
FUNCTION USINT_TO_SINT : SINT
VAR_INPUT
	in : USINT;
END_VAR
	USINT_TO_SINT := in;
END_FUNCTION

(********************
*
* Converts USINT to ULINT
*
*********************)
FUNCTION USINT_TO_ULINT : ULINT
VAR_INPUT
	in : USINT;
END_VAR
	USINT_TO_ULINT := in;
END_FUNCTION

(********************
*
* Converts USINT to UDINT
*
*********************)
FUNCTION USINT_TO_UDINT : UDINT
VAR_INPUT
	in : USINT;
END_VAR
	USINT_TO_UDINT := in;
END_FUNCTION

(********************
*
* Converts USINT to UINT
*
*********************)
FUNCTION USINT_TO_UINT : UINT
VAR_INPUT
	in : USINT;
END_VAR
	USINT_TO_UINT := in;
END_FUNCTION

(* ---- string_conversion.st ---- *)
(********************
*
* Converts WSTRING to STRING
* Will return a STRING with default length of 81
*
*********************)
{external}
FUNCTION WSTRING_TO_STRING : STRING
VAR_INPUT {ref}
	in : WSTRING;
END_VAR
END_FUNCTION

(********************
*
* Converts WSTRING to WCHAR
*
*********************)
FUNCTION WSTRING_TO_WCHAR : WCHAR
VAR_INPUT {ref}
	in : WSTRING;
END_VAR
VAR
	ptr : REF_TO WCHAR;
END_VAR
	ptr := &in;
	WSTRING_TO_WCHAR := ptr^;
END_FUNCTION

(********************
*
* Converts STRING to WSTRING
* Will return a WSTRING with default length of 81
*
*********************)
{external}
FUNCTION STRING_TO_WSTRING : WSTRING
VAR_INPUT {ref}
	in : STRING;
END_VAR
END_FUNCTION

(********************
*
* Converts STRING to CHAR
*
*********************)
FUNCTION STRING_TO_CHAR : CHAR
VAR_INPUT {ref}
	in : STRING;
END_VAR
VAR
	ptr : REF_TO CHAR;
END_VAR
	ptr := &in;
	STRING_TO_CHAR := ptr^;
END_FUNCTION

(********************
*
* Converts WCHAR to WSTRING
*
*********************)
FUNCTION WCHAR_TO_WSTRING : WSTRING
VAR_INPUT
	in : WCHAR;
END_VAR
VAR
	ptr : REF_TO WSTRING;
END_VAR
	ptr := &in;
	WCHAR_TO_WSTRING := ptr^;
END_FUNCTION

(********************
*
* Converts WCHAR to CHAR
*
*********************)
{external}
FUNCTION WCHAR_TO_CHAR : CHAR
VAR_INPUT
	in : WCHAR;
END_VAR
END_FUNCTION

(********************
*
* Converts CHAR to STRING
*
*********************)
FUNCTION CHAR_TO_STRING : STRING
VAR_INPUT
	in : CHAR;
END_VAR
VAR
	ptr : REF_TO STRING;
END_VAR
	ptr := &in;
	CHAR_TO_STRING := ptr^;
END_FUNCTION

(********************
*
* Converts CHAR to WCHAR
*
*********************)
{external}
FUNCTION CHAR_TO_WCHAR : WCHAR
VAR_INPUT
	in : CHAR;
END_VAR
END_FUNCTION

(* ---- string_functions.st ---- *)
(******************************************************************************
Description: String length
Input:
    - IN:   A character string
Return: String length
******************************************************************************)
{external}
FUNCTION LEN <T: ANY_STRING> : DINT
VAR_INPUT {ref}
	IN : T;
END_VAR
END_FUNCTION

(******************************************************************************
Description: Left
Input:
    - IN:   A character string
    - L:    The length of the substring
Return: A substring consisting of the leftmost L characters of IN
******************************************************************************)
FUNCTION LEFT <T: ANY_STRING> : T
VAR_INPUT {ref}
	IN : T;
END_VAR
VAR_INPUT
    L  : DINT;
END_VAR
END_FUNCTION

{external}
FUNCTION LEFT_EXT<T: ANY_STRING> : DINT
VAR_INPUT {ref}
	IN : T;
END_VAR
VAR_INPUT
    L  : DINT;
END_VAR
VAR_IN_OUT
    OUT: T;
END_VAR
END_FUNCTION

FUNCTION LEFT__STRING : STRING[2048]
VAR_INPUT {ref}
	IN : STRING[2048];
END_VAR
VAR_INPUT
    L  : DINT;
END_VAR
    LEFT_EXT(IN, L, LEFT__STRING);
END_FUNCTION

FUNCTION LEFT__WSTRING : WSTRING[2048]
VAR_INPUT {ref}
	IN : WSTRING[2048];
END_VAR
VAR_INPUT
    L  : DINT;
END_VAR
    LEFT_EXT(IN, L, LEFT__WSTRING);
END_FUNCTION

{external}
FUNCTION LEFT_EXT__STRING : DINT
VAR_INPUT {ref}
	IN : STRING[2048];
END_VAR
VAR_INPUT
    L  : DINT;
END_VAR
VAR_IN_OUT
    OUT: STRING[2048];
END_VAR
END_FUNCTION

{external}
FUNCTION LEFT_EXT__WSTRING : DINT
VAR_INPUT {ref}
	IN : WSTRING[2048];
END_VAR
VAR_INPUT
    L  : DINT;
END_VAR
VAR_IN_OUT
    OUT: WSTRING[2048];
END_VAR
END_FUNCTION

(******************************************************************************
Description: Right
Input:
    - IN:   A character string
    - L:    The length of the substring
Return: A substring consisting of the rightmost L characters of IN
******************************************************************************)
FUNCTION RIGHT <T: ANY_STRING> : T
VAR_INPUT {ref}
	IN : T;
END_VAR
VAR_INPUT
    L  : DINT;
END_VAR
END_FUNCTION

{external}
FUNCTION RIGHT_EXT<T: ANY_STRING> : DINT
VAR_INPUT {ref}
	IN : T;
END_VAR
VAR_INPUT
    L  : DINT;
END_VAR
VAR_IN_OUT
    OUT: T;
END_VAR
END_FUNCTION

FUNCTION RIGHT__STRING : STRING[2048]
VAR_INPUT {ref}
	IN : STRING[2048];
END_VAR
VAR_INPUT
    L  : DINT;
END_VAR
    RIGHT_EXT(IN, L, RIGHT__STRING);
END_FUNCTION

FUNCTION RIGHT__WSTRING : WSTRING[2048]
VAR_INPUT {ref}
	IN : WSTRING[2048];
END_VAR
VAR_INPUT
    L  : DINT;
END_VAR
    RIGHT_EXT(IN, L, RIGHT__WSTRING);
END_FUNCTION

{external}
FUNCTION RIGHT_EXT__STRING : DINT
VAR_INPUT {ref}
	IN : STRING[2048];
END_VAR
VAR_INPUT
    L  : DINT;
END_VAR
VAR_IN_OUT
    OUT: STRING[2048];
END_VAR
END_FUNCTION

{external}
FUNCTION RIGHT_EXT__WSTRING : DINT
VAR_INPUT {ref}
	IN : WSTRING[2048];
END_VAR
VAR_INPUT
    L  : DINT;
END_VAR
VAR_IN_OUT
    OUT: WSTRING[2048];
END_VAR
END_FUNCTION

(******************************************************************************
Description: Middle
Input:
    - IN:   A character string
    - L:    The length of the substring
    - P:    The starting index position
Return:
    A substring that contains L characters starting
    from position P in a string.
******************************************************************************)
FUNCTION MID <T: ANY_STRING> : T
VAR_INPUT {ref}
	IN : T;
END_VAR
VAR_INPUT
    L  : DINT;
    P  : DINT;
END_VAR
END_FUNCTION

{external}
FUNCTION MID_EXT<T: ANY_STRING> : DINT
VAR_INPUT {ref}
	IN : T;
END_VAR
VAR_INPUT
    L  : DINT;
    P  : DINT;
END_VAR
VAR_IN_OUT
    OUT: T;
END_VAR
END_FUNCTION

FUNCTION MID__STRING : STRING[2048]
VAR_INPUT {ref}
	IN : STRING[2048];
END_VAR
VAR_INPUT
    L  : DINT;
    P  : DINT;
END_VAR
    MID_EXT(IN, L, P, MID__STRING);
END_FUNCTION

FUNCTION MID__WSTRING : WSTRING[2048]
VAR_INPUT {ref}
	IN : WSTRING[2048];
END_VAR
VAR_INPUT
    L  : DINT;
    P  : DINT;
END_VAR
    MID_EXT(IN, L, P, MID__WSTRING);
END_FUNCTION

{external}
FUNCTION MID_EXT__STRING : DINT
VAR_INPUT {ref}
	IN : STRING[2048];
END_VAR
VAR_INPUT
    L  : DINT;
    P  : DINT;
END_VAR
VAR_IN_OUT
    OUT: STRING[2048];
END_VAR
END_FUNCTION

{external}
FUNCTION MID_EXT__WSTRING : DINT
VAR_INPUT {ref}
	IN : WSTRING[2048];
END_VAR
VAR_INPUT
    L  : DINT;
    P  : DINT;
END_VAR
VAR_IN_OUT
    OUT: WSTRING[2048];
END_VAR
END_FUNCTION

(******************************************************************************
Description: Extensible concatenation
Input:
    - IN:   Two or more comma-separated strings
Return:
    A string combining all given input strings in the same order
    as the given string parameters.
******************************************************************************)
{external}
FUNCTION CONCAT <T: ANY_STRING> : T
VAR_INPUT {ref}
	args : {sized} T...;
END_VAR
END_FUNCTION

{external}
FUNCTION CONCAT_EXT<T: ANY_STRING> : DINT
VAR_IN_OUT
    OUT: T;
END_VAR
VAR_INPUT {ref}
    args: {sized} T...;
END_VAR
END_FUNCTION

(******************************************************************************
Description: Insert
Input:
    IN1:    The string to insert into
    IN2:    The string to insert
    P:      The position at which to insert
Return:
    A string consisting of IN2 inserted at position P into string IN1
******************************************************************************)
FUNCTION INSERT <T: ANY_STRING> : T
VAR_INPUT {ref}
	IN1 : T;
    IN2 : T;
END_VAR
VAR_INPUT
    P   : DINT;
END_VAR
END_FUNCTION

{external}
FUNCTION INSERT_EXT<T: ANY_STRING> : DINT
VAR_INPUT {ref}
	IN1 : T;
    IN2 : T;
END_VAR
VAR_INPUT
    P   : DINT;
END_VAR
VAR_IN_OUT
    OUT: T;
END_VAR
END_FUNCTION

FUNCTION INSERT__STRING : STRING[2048]
VAR_INPUT {ref}
	IN1 : STRING[2048];
    IN2 : STRING[2048];
END_VAR
VAR_INPUT
    P   : DINT;
END_VAR
    INSERT_EXT(IN1, IN2, P, INSERT__STRING);
END_FUNCTION

FUNCTION INSERT__WSTRING : WSTRING[2048]
VAR_INPUT {ref}
	IN1 : WSTRING[2048];
    IN2 : WSTRING[2048];
END_VAR
VAR_INPUT
    P   : DINT;
END_VAR
    INSERT_EXT(IN1, IN2, P, INSERT__WSTRING);
END_FUNCTION

{external}
FUNCTION INSERT_EXT__STRING : DINT
VAR_INPUT {ref}
	IN1 : STRING[2048];
    IN2 : STRING[2048];
END_VAR
VAR_INPUT
    P   : DINT;
END_VAR
VAR_IN_OUT
    OUT: STRING[2048];
END_VAR
END_FUNCTION

{external}
FUNCTION INSERT_EXT__WSTRING : DINT
VAR_INPUT {ref}
	IN1 : WSTRING[2048];
    IN2 : WSTRING[2048];
END_VAR
VAR_INPUT
    P   : DINT;
END_VAR
VAR_IN_OUT
    OUT: WSTRING[2048];
END_VAR
END_FUNCTION

(******************************************************************************
Description: Delete
Input:
Return:
******************************************************************************)
FUNCTION DELETE <T: ANY_STRING> : T
VAR_INPUT {ref}
	IN : T;
END_VAR
VAR_INPUT
    L  : DINT;
    P  : DINT;
END_VAR
END_FUNCTION

{external}
FUNCTION DELETE_EXT<T: ANY_STRING> : DINT
VAR_INPUT {ref}
	IN : T;
END_VAR
VAR_INPUT
    L  : DINT;
    P  : DINT;
END_VAR
VAR_IN_OUT
    OUT: T;
END_VAR
END_FUNCTION

FUNCTION DELETE__STRING : STRING[2048]
VAR_INPUT {ref}
	IN : STRING[2048];
END_VAR
VAR_INPUT
    L  : DINT;
    P  : DINT;
END_VAR
    DELETE_EXT(IN, L, P, DELETE__STRING);
END_FUNCTION

FUNCTION DELETE__WSTRING : WSTRING[2048]
VAR_INPUT {ref}
	IN : WSTRING[2048];
END_VAR
VAR_INPUT
    L  : DINT;
    P  : DINT;
END_VAR
    DELETE_EXT(IN, L, P, DELETE__WSTRING);
END_FUNCTION

{external}
FUNCTION DELETE_EXT__STRING : DINT
VAR_INPUT {ref}
	IN : STRING[2048];
END_VAR
VAR_INPUT
    L  : DINT;
    P  : DINT;
END_VAR
VAR_IN_OUT
    OUT: STRING[2048];
END_VAR
END_FUNCTION

{external}
FUNCTION DELETE_EXT__WSTRING : DINT
VAR_INPUT {ref}
	IN : WSTRING[2048];
END_VAR
VAR_INPUT
    L  : DINT;
    P  : DINT;
END_VAR
VAR_IN_OUT
    OUT: WSTRING[2048];
END_VAR
END_FUNCTION
(******************************************************************************
Description: Replace
Input:
Return:
******************************************************************************)
FUNCTION REPLACE <T: ANY_STRING> : T
VAR_INPUT {ref}
	IN1 : T;
    IN2 : T;
END_VAR
VAR_INPUT
    L  : DINT;
    P  : DINT;
END_VAR
END_FUNCTION

{external}
FUNCTION REPLACE_EXT <T: ANY_STRING> : DINT
VAR_INPUT {ref}
    IN1 : T;
    IN2 : T;
END_VAR
VAR_INPUT
    L   : DINT;
    P   : DINT;
END_VAR
VAR_IN_OUT
    OUT : T;
END_VAR
END_FUNCTION

FUNCTION REPLACE__STRING : STRING[2048]
VAR_INPUT {ref}
	IN1 : STRING[2048];
    IN2 : STRING[2048];
END_VAR
VAR_INPUT
    L  : DINT;
    P  : DINT;
END_VAR
    REPLACE_EXT(IN1, IN2, L, P, REPLACE__STRING);
END_FUNCTION

FUNCTION REPLACE__WSTRING : WSTRING[2048]
VAR_INPUT {ref}
    IN1 : WSTRING[2048];
    IN2 : WSTRING[2048];
END_VAR
VAR_INPUT
    L   : DINT;
    P   : DINT;
END_VAR
    REPLACE_EXT(IN1, IN2, L, P, REPLACE__WSTRING);
END_FUNCTION

{external}
FUNCTION REPLACE_EXT__STRING : DINT
VAR_INPUT {ref}
    IN1 : STRING[2048];
    IN2 : STRING[2048];
END_VAR
VAR_INPUT
    L   : DINT;
    P   : DINT;
END_VAR
VAR_IN_OUT
    OUT : STRING[2048];
END_VAR
END_FUNCTION

{external}
FUNCTION REPLACE_EXT__WSTRING : DINT
VAR_INPUT {ref}
    IN1 : WSTRING[2048];
    IN2 : WSTRING[2048];
END_VAR
VAR_INPUT
    L   : DINT;
    P   : DINT;
END_VAR
VAR_IN_OUT
    OUT : WSTRING[2048];
END_VAR
END_FUNCTION

(******************************************************************************
Description: Find
Input:
Return:
******************************************************************************)
{external}
FUNCTION FIND <T: ANY_STRING> : DINT
VAR_INPUT {ref}
	IN1 : T;
    IN2 : T;
END_VAR
END_FUNCTION

(******************************************************************************
Description: Decreasing sequence
Input:
Return:
******************************************************************************)
{external}
FUNCTION GT <T: ANY_STRING> : BOOL
VAR_INPUT {ref}
	IN1 : {sized} T...;
END_VAR
END_FUNCTION

(******************************************************************************
Description: Monotonic sequence
Input:
Return:
******************************************************************************)
{external}
FUNCTION GE <T: ANY_STRING> : BOOL
VAR_INPUT {ref}
	IN1 : {sized} T...;
END_VAR
END_FUNCTION

(******************************************************************************
Description: Equality
Input:
Return:
******************************************************************************)
{external}
FUNCTION EQ <T: ANY_STRING> : BOOL
VAR_INPUT {ref}
	IN1 : {sized} T...;
END_VAR
END_FUNCTION

(******************************************************************************
Description: Monotonic sequence
Input:
Return:
******************************************************************************)
{external}
FUNCTION LE <T: ANY_STRING> : BOOL
VAR_INPUT {ref}
	IN1 : {sized} T...;
END_VAR
END_FUNCTION

(******************************************************************************
Description: Increasing sequence
Input:
Return:
******************************************************************************)
{external}
FUNCTION LT <T: ANY_STRING> : BOOL
VAR_INPUT {ref}
	IN1 : {sized} T...;
END_VAR
END_FUNCTION

(******************************************************************************
Description: Inequality
Input:
Return:
******************************************************************************)
{external}
FUNCTION NE <T: ANY_STRING> : BOOL
VAR_INPUT {ref}
	IN1 : T;
    IN2 : T;
END_VAR
END_FUNCTION
